// TIA Portal V19 program export: 12 tag tables, 4 data types, 5 data blocks, 16 code blocks (in call order from the OBs), 12 instance data blocks

VAR_GLOBAL   // PLC tag table "Default tag table"
   FirstScan AT %M101.0 : Bool;
   DiagStatusUpdate AT %M101.1 : Bool;
   AlwaysTRUE AT %M101.2 : Bool;
   AlwaysFALSE AT %M101.3 : Bool;
   System_Byte AT %MB101 : Byte;
   Clock_Byte AT %MB100 : Byte;
   Clock_10Hz AT %M100.0 : Bool;
   Clock_5Hz AT %M100.1 : Bool;
   "Clock_2.5Hz" AT %M100.2 : Bool;
   Clock_2Hz AT %M100.3 : Bool;
   "Clock_1.25Hz" AT %M100.4 : Bool;
   Clock_1Hz AT %M100.5 : Bool;
   "Clock_0.625Hz" AT %M100.6 : Bool;
   "Clock_0.5Hz" AT %M100.7 : Bool;
END_VAR

VAR_GLOBAL   // PLC tag table "DemoCaseTags"
   POT4_G120 AT %MD30 : Real;
   HMI_IO_Test AT %M10.4 : Bool;
   PB_Green_1200 AT %M60.0 : Bool;
   PB_Blue_1200 AT %M60.1 : Bool;
   POT3_Upper_1200 AT %MW62 : Int;
   PB_Green_Lamp_1200 AT %M64.0 : Bool;
   PB_Blue_Lamp_1200 AT %M64.1 : Bool;
   TopLights_Green_1200 AT %M64.5 : Bool;
   TopLights_Red_1200 AT %M64.6 : Bool;
   TopLights_Blue_1200 AT %M64.7 : Bool;
   "1200_Inputs" AT %MB60 : Byte;
   "1200_Outputs" AT %MB64 : Byte;
   "1200_All_Inputs" AT %MD60 : DWord;
   OS6 AT %M11.4 : Bool;
   "Red Latch" AT %M11.5 : Bool;
   "Green Latch" AT %M11.6 : Bool;
   GateClosed AT %M11.7 : Bool;
   "Blue Latch" AT %M20.3 : Bool;
   Coordination AT %MW36 : Int;
   POT2_Warning AT %M20.4 : Bool;
END_VAR

VAR_GLOBAL   // PLC tag table "HMIConveyor"
   ConveyorOn AT %M10.0 : Bool;
   ConveyorMoving AT %M10.1 : Bool;
   Conveyor_MPM AT %MW12 : Int;
   Conveyor_Max_MPM AT %MW14 : Int;
   Start_System_HMI AT %M20.0 : Bool;
   Stop_System_HMI AT %M20.1 : Bool;
   Reset_System_HMI AT %M20.2 : Bool;
   OS1 AT %M10.2 : Bool;
   ARM_MPM AT %MW34 : Int;
   OS11 AT %M74.3 : Bool;
END_VAR

VAR_GLOBAL   // PLC tag table "KP8Tags"
   Toggle_Switch2 AT %M50.0 : Bool;   // KP8 bit that is toggled each time is pressed
   HMI_KP8_JogFwd AT %M50.1 : Bool;
   HMI_KP8_Stop AT %M50.2 : Bool;
   Toggle_Switch1 AT %M50.4 : Bool;   // KP8 bit that is toggled each time is pressed
   HMI_KP8_JogRev AT %M50.5 : Bool;
   HMI_KP8_Start AT %M50.6 : Bool;
   Toggle_Enable_Disable AT %M50.7 : Bool;   // KP8 bit that is toggled each time is pressed
   HMI_KP8_Red AT %MB70 : Byte;
   HMI_KP8_Green AT %MB71 : Byte;
   HMI_KP8_Blue AT %MB72 : Byte;
   HMI_KP8_Enable_Disable AT %M73.0 : Bool;
   HMI_KP8_Reset AT %M73.1 : Bool;
   HMI_KP8_Switch1 AT %M73.2 : Bool;
   HMI_KP8_Switch2 AT %M73.3 : Bool;
   OS8 AT %M74.0 : Bool;
   OS9 AT %M74.1 : Bool;
   OS10 AT %M74.2 : Bool;
END_VAR

VAR_GLOBAL   // PLC tag table "SafetyTags"
   Safety_PB_Blue_Lamp AT %M90.0 : Bool;
END_VAR

VAR_GLOBAL   // PLC tag table "Speed Control"
   POT2_Lower_Real AT %MD38 : Real;
   Tmp AT %MW4 : Word;
   POT1_Upper__Real AT %MD16 : Real;
   MyIndex AT %MW6 : Int;
   Drive_Error AT %M11.3 : Bool;
   OS2 AT %M10.3 : Bool;
   OS3 AT %M10.5 : Bool;
   G120_Error AT %M10.6 : Bool;
   G120_Enabled AT %M10.7 : Bool;
   G120_Run_Velocity AT %M11.0 : Bool;
   OS4 AT %M11.1 : Bool;
   OS5 AT %M11.2 : Bool;
   BusyMV AT %M0.0 : Bool;
   OS7 AT %M21.3 : Bool;
   ConveyorWorking AT %M6.0 : Bool;   // Conveyor Diagnostic Tag
END_VAR

VAR_GLOBAL   // PLC tag table "Encoder"
END_VAR

VAR_GLOBAL   // PLC tag table "G120"
   SpeedAxis_1_Actor_Interface_AddressIn AT %I256.0 : "PD_TEL1_IN";
   SpeedAxis_1_Actor_Interface_AddressOut AT %Q256.0 : "PD_TEL1_OUT";
END_VAR

VAR_GLOBAL   // PLC tag table "KP8"
   Jog_Reverse_Green_KP8 AT %Q51.5 : Bool;   // KP8
   Enable_Disable_KP8 AT %I50.7 : Bool;   // KP8
   Drive_Start_KP8 AT %I50.6 : Bool;   // KP8
   Jog_Reverse_KP8 AT %I50.5 : Bool;   // KP8
   Switch1_KP8 AT %I50.4 : Bool;   // KP8
   Enable_Disable_Green_KP8 AT %Q51.7 : Bool;   // KP8
   Drive_Start_Red_KP8 AT %Q50.6 : Bool;   // KP8
   Jog_Reverse_Red_KP8 AT %Q50.5 : Bool;   // KP8
   Switch1_Red_KP8 AT %Q50.4 : Bool;   // KP8
   RESET_KP8 AT %I50.3 : Bool;   // KP8
   Drive_Stop_KP8 AT %I50.2 : Bool;   // KP8
   Jog_Forward_KP8 AT %I50.1 : Bool;   // KP8
   RESET_Red_KP8 AT %Q50.3 : Bool;   // KP8
   Drive_Stop_Red_KP8 AT %Q50.2 : Bool;   // KP8
   Jog_Forward_Red_KP8 AT %Q50.1 : Bool;   // KP8
   Switch2_KP8 AT %I50.0 : Bool;   // KP8
   Switch2_Red_KP8 AT %Q50.0 : Bool;   // KP8
   Enable_Disable_Red_KP8 AT %Q50.7 : Bool;   // KP8
   Drive_Start_Green_KP8 AT %Q51.6 : Bool;   // KP8
   Switch1_Green_KP8 AT %Q51.4 : Bool;   // KP8
   RESET_Green_KP8 AT %Q51.3 : Bool;   // KP8
   Drive_Stop_Green_KP8 AT %Q51.2 : Bool;   // KP8
   Jog_Forward_Green_KP8 AT %Q51.1 : Bool;   // KP8
   Switch2_Green_KP8 AT %Q51.0 : Bool;   // KP8
   Switch2_Blue_KP8 AT %Q52.0 : Bool;   // KP8
   Jog_Forward_Blue_KP8 AT %Q52.1 : Bool;   // KP8
   Drive_Stop_Blue_KP8 AT %Q52.2 : Bool;   // KP8
   RESET_Blue_KP8 AT %Q52.3 : Bool;   // KP8
   Switch1_Blue_KP8 AT %Q52.4 : Bool;   // KP8
   Jog_Reverse_Blue_KP8 AT %Q52.5 : Bool;   // KP8
   Drive_Start_Blue_KP8 AT %Q52.6 : Bool;   // KP8
   Enable_Disable_Blue_KP8 AT %Q52.7 : Bool;   // KP8
   KP8_Red AT %QB50 : Byte;   // KP8
   KP8_Green AT %QB51 : Byte;   // KP8
   KP8_Blue AT %QB52 : Byte;   // KP8
END_VAR

VAR_GLOBAL   // PLC tag table "LocalMP"
   PB_Green_1500 AT %I0.0 : Bool;
   PB_Blue_1500 AT %I0.1 : Bool;
   POT1_Upper_1500 AT %IW6 : Int;   // connected to AI channel 2
   POT2_Lower_1500 AT %IW14 : Int;   // connected to AI channel 6
END_VAR

VAR_GLOBAL   // PLC tag table "RemoteSP"
   PB_Green_Lamp AT %Q8.0 : Bool;
   PB_Blue_Lamp AT %Q8.1 : Bool;
   TopLights_green_1500 AT %Q10.0 : Bool;   // TopLight green 1=on 0=off
   TopLights_red_1500 AT %Q10.1 : Bool;   // TopLight red 1=on 0=off
   TopLights_blue_1500 AT %Q10.2 : Bool;   // TopLight blue 1=on 0=off
   "ESTOP CH1" AT %I18.1 : Bool;
   Estop_LED AT %Q24.0 : Bool;
   "RFID_Gate CH1" AT %I18.0 : Bool;
   RFID_Gate_AUX AT %I22.2 : Bool;
END_VAR

VAR_GLOBAL   // PLC tag table "S71200IDevice"
   "Out to 1200" AT %QW100 : Int;
   PB_Green_from_1200 AT %I100.0 : Bool;
   PB_Blue_from_1200 AT %I100.1 : Bool;
   POT_from_1200 AT %IW102 : Word;
END_VAR

TYPE "HEADER"
   STRUCT
      REQ_REF : Byte;
      REQ_ID : Byte;
      AXIS : Byte;
      NO_PARAM : Byte;
   END_STRUCT;
END_TYPE

TYPE "PARAMETERADDR"
   STRUCT
      ATTRIBUTE : Byte;
      NO_ELEM : Byte;
      PARA_NO : Word;
      SUBINDEX : Word;
   END_STRUCT;
END_TYPE

TYPE "SiemensDataType"
   STRUCT
      Test1 : Bool;
      Test2 : Bool;
      Test3 : Bool;
      Test4 : Bool;
      Test5 : Bool;
      Test6 : Bool;
      Test7 : Bool;
   END_STRUCT;
END_TYPE

TYPE "Time Zone"
   STRUCT
      City : String;
      "Local Time" : Time_Of_Day;
      Offset : Time;
   END_STRUCT;
END_TYPE

DATA_BLOCK "GlobalDB"   // DB2
{ S7_Optimized_Access := 'TRUE' }
// stored: MemoryReserve 100
   VAR
      TagData : "SiemensDataType";
   END_VAR
BEGIN
END_DATA_BLOCK

DATA_BLOCK "GraphicsData"   // DB1
{ S7_Optimized_Access := 'TRUE' }
// stored: MemoryReserve 100
   VAR
      HMI_Graphic_Index : Int;
      HMI_Box_Cnt : DInt;
      HMI_Pallet_Cnt : DInt;
   END_VAR
BEGIN
END_DATA_BLOCK

DATA_BLOCK "TimeZones"   // DB13
{ S7_Optimized_Access := 'TRUE' }
// stored: MemoryReserve 100
   VAR
      UTC_0 : "Time Zone";
      UTC_1 { S7_SetPoint := 'True'} : "Time Zone";
      UTC_2 { S7_SetPoint := 'True'} : "Time Zone";
   END_VAR
BEGIN
   UTC_0.City := 'London';
   UTC_0.Offset := T#0H;
   UTC_1.City := 'Berlin';
   UTC_1.Offset := T#1H;
   UTC_2.City := 'Cairo';
   UTC_2.Offset := T#2H;
END_DATA_BLOCK

DATA_BLOCK "TestInterConnLPythagorean"   // DB10001
{ S7_Optimized_Access := 'TRUE' }
// #@AutoGenerated
// stored: MemoryReserve 100
   VAR
      "a" : Real;
      "b" : Real;
      c : Real;
      valid : Bool;
   END_VAR
BEGIN
END_DATA_BLOCK

DATA_BLOCK "Connect_DB"   // DB7
{ S7_Optimized_Access := 'TRUE' }
// stored: MemoryReserve 100
   VAR
      "Out to 1200" : Int;
   END_VAR
BEGIN
END_DATA_BLOCK

ORGANIZATION_BLOCK "Main"   // OB1, LAD, ProgramCycle
TITLE = "Main Program Sweep (Cycle)"
{ S7_Optimized_Access := 'TRUE' }
// TIA Demo Project
// 1500 password is Siemens1
// stored: SetENOAutomatically false
   VAR_INPUT
      Initial_Call : Bool;   // Initial call of this OB
      Remanence : Bool;   // =True, if remanent data are available
   END_VAR
   VAR_TEMP   // added for the SCL form of the ladder/FBD networks
      _w1 : Bool;
      _w2 : Bool;
   END_VAR
BEGIN

REGION Network 1: Scale the Potentiometer raw value to a Real between 0.0-1500.0
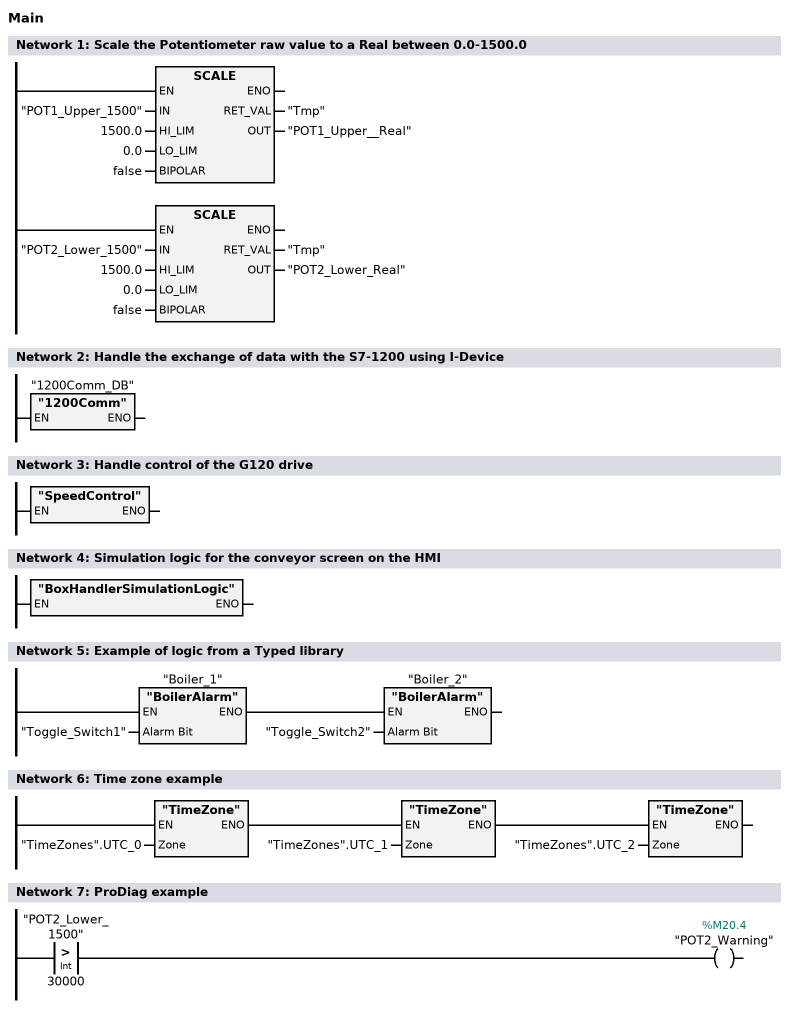
   "Tmp" := SCALE(IN := "POT1_Upper_1500",
                  HI_LIM := 1500.0,
                  LO_LIM := 0.0,
                  BIPOLAR := false,
                  OUT => "POT1_Upper__Real");
   "Tmp" := SCALE(IN := "POT2_Lower_1500",
                  HI_LIM := 1500.0,
                  LO_LIM := 0.0,
                  BIPOLAR := false,
                  OUT => "POT2_Lower_Real");
END_REGION

REGION Network 2: Handle the exchange of data with the S7-1200 using I-Device
   RUNG wire#powerrail
      "1200Comm_DB"()
   END_RUNG
   // the same network as SCL:
   "1200Comm_DB"();   // "1200Comm"
END_REGION

REGION Network 3: Handle control of the G120 drive
   RUNG wire#powerrail
      "SpeedControl"()
   END_RUNG
   // the same network as SCL:
   "SpeedControl"();
END_REGION

REGION Network 4: Simulation logic for the conveyor screen on the HMI
   RUNG wire#powerrail
      "BoxHandlerSimulationLogic"()
   END_RUNG
   // the same network as SCL:
   "BoxHandlerSimulationLogic"();
END_REGION

REGION Network 5: Example of logic from a Typed library
   RUNG wire#powerrail
      "Boiler_1"("Alarm Bit" := "Toggle_Switch1")
      "Boiler_2"("Alarm Bit" := "Toggle_Switch2")
   END_RUNG
   // the same network as SCL:
   "Boiler_1"("Alarm Bit" := "Toggle_Switch1", ENO => #_w1);   // "BoilerAlarm"
   IF #_w1 THEN
       "Boiler_2"("Alarm Bit" := "Toggle_Switch2");   // "BoilerAlarm"
   END_IF;
END_REGION

REGION Network 6: Time zone example
   RUNG wire#powerrail
      "TimeZone"(Zone := "TimeZones".UTC_0)
      "TimeZone"(Zone := "TimeZones".UTC_1)
      "TimeZone"(Zone := "TimeZones".UTC_2)
   END_RUNG
   // the same network as SCL:
   "TimeZone"(Zone := "TimeZones".UTC_0, ENO => #_w1);
   "TimeZone"(EN := #_w1, Zone := "TimeZones".UTC_1, ENO => #_w2);
   IF #_w2 THEN "TimeZone"(Zone := "TimeZones".UTC_2); END_IF;
END_REGION

REGION Network 7: ProDiag example
   RUNG wire#powerrail
      { S7_Templates := "SrcType := Int" } GT_Contact(in1 := "POT2_Lower_1500", in2 := 30000)
      Coil( "POT2_Warning" )
   END_RUNG
   // the same network as SCL:
   "POT2_Warning" := "POT2_Lower_1500" > 30000;
END_REGION
END_ORGANIZATION_BLOCK

FUNCTION_BLOCK "1200Comm"   // FB3, LAD
TITLE = I Device exchange of data with the S7-1200
{ S7_Optimized_Access := 'TRUE' }
// stored: MemoryReserve 100, SetENOAutomatically false
BEGIN

REGION Network 1: Pass light data to the 1200
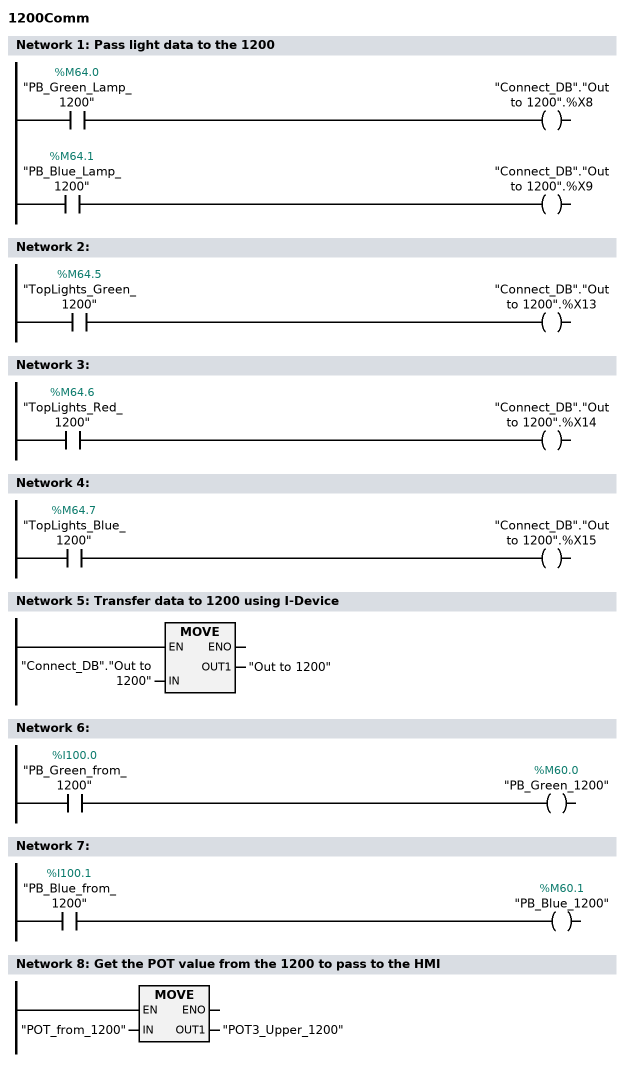
   RUNG wire#powerrail
      Contact( "PB_Green_Lamp_1200" )
      Coil( "Connect_DB"."Out to 1200".%X8 )
   END_RUNG
   RUNG wire#powerrail
      Contact( "PB_Blue_Lamp_1200" )
      Coil( "Connect_DB"."Out to 1200".%X9 )
   END_RUNG
   // the same network as SCL:
   "Connect_DB"."Out to 1200".%X8 := "PB_Green_Lamp_1200";
   "Connect_DB"."Out to 1200".%X9 := "PB_Blue_Lamp_1200";
END_REGION

REGION Network 2
   RUNG wire#powerrail
      Contact( "TopLights_Green_1200" )
      Coil( "Connect_DB"."Out to 1200".%X13 )
   END_RUNG
   // the same network as SCL:
   "Connect_DB"."Out to 1200".%X13 := "TopLights_Green_1200";
END_REGION

REGION Network 3
   RUNG wire#powerrail
      Contact( "TopLights_Red_1200" )
      Coil( "Connect_DB"."Out to 1200".%X14 )
   END_RUNG
   // the same network as SCL:
   "Connect_DB"."Out to 1200".%X14 := "TopLights_Red_1200";
END_REGION

REGION Network 4
   RUNG wire#powerrail
      Contact( "TopLights_Blue_1200" )
      Coil( "Connect_DB"."Out to 1200".%X15 )
   END_RUNG
   // the same network as SCL:
   "Connect_DB"."Out to 1200".%X15 := "TopLights_Blue_1200";
END_REGION

REGION Network 5: Transfer data to 1200 using I-Device
   RUNG wire#powerrail
      Move(in := "Connect_DB"."Out to 1200", out1 => "Out to 1200")
   END_RUNG
   // the same network as SCL:
   "Out to 1200" := "Connect_DB"."Out to 1200";
END_REGION

REGION Network 6
   RUNG wire#powerrail
      Contact( "PB_Green_from_1200" )
      Coil( "PB_Green_1200" )
   END_RUNG
   // the same network as SCL:
   "PB_Green_1200" := "PB_Green_from_1200";
END_REGION

REGION Network 7
   RUNG wire#powerrail
      Contact( "PB_Blue_from_1200" )
      Coil( "PB_Blue_1200" )
   END_RUNG
   // the same network as SCL:
   "PB_Blue_1200" := "PB_Blue_from_1200";
END_REGION

REGION Network 8: Get the POT value from the 1200 to pass to the HMI
   RUNG wire#powerrail
      Move(in := "POT_from_1200", out1 => "POT3_Upper_1200")
   END_RUNG
   // the same network as SCL:
   "POT3_Upper_1200" := "POT_from_1200";
END_REGION
END_FUNCTION_BLOCK

FUNCTION "SpeedControl" : Void   // FC1, LAD
TITLE = G120 drive Control
{ S7_Optimized_Access := 'TRUE' }
// stored: SetENOAutomatically false
   VAR_TEMP   // added for the SCL form of the ladder/FBD networks
      _w1 : Bool;
      _w2 : Bool;
   END_VAR
BEGIN

REGION Network 1: Enable the G120
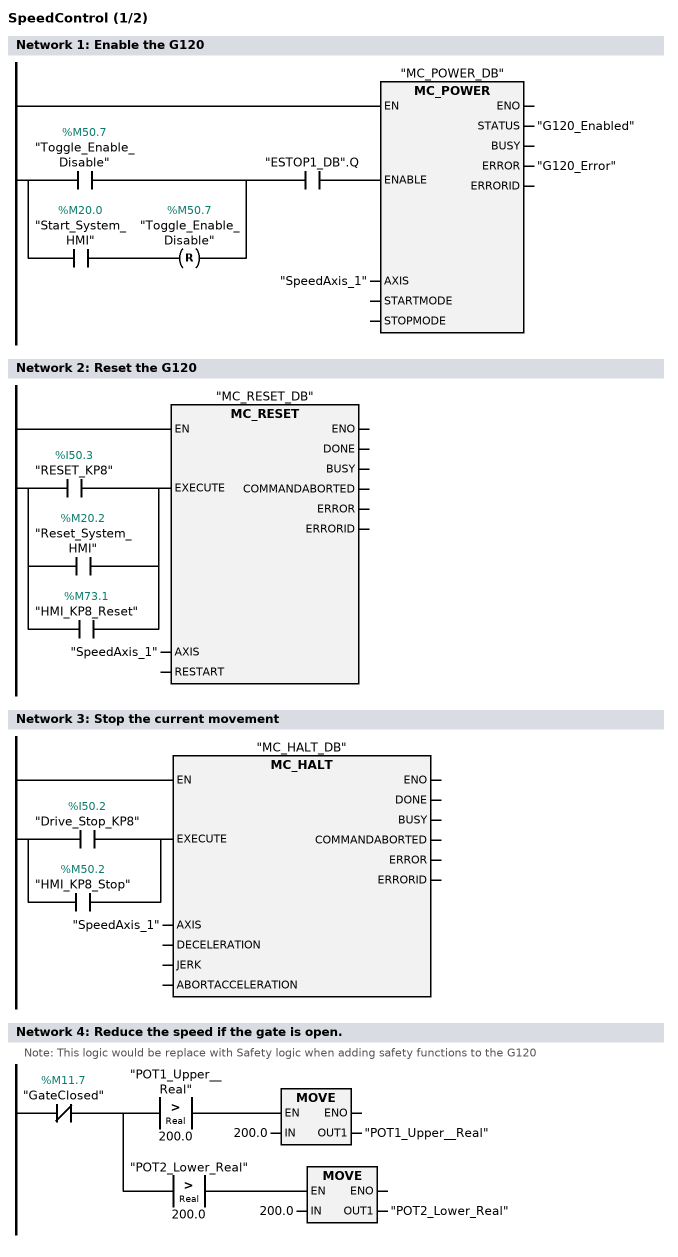
   RUNG wire#powerrail
      "MC_POWER_DB".MC_POWER(Enable := wire#w2, Axis := "SpeedAxis_1", StartMode :=, StopMode :=, Status => "G120_Enabled", Busy =>, Error => "G120_Error", ErrorId =>)
   END_RUNG
   RUNG wire#powerrail
      Contact( "Toggle_Enable_Disable" )
      wire#w1
      Contact( "ESTOP1_DB".Q )
   END_RUNG wire#w2
   RUNG wire#powerrail
      Contact( "Start_System_HMI" )
      R_Coil( "Toggle_Enable_Disable" )
   END_RUNG wire#w1
   // the same network as SCL:
   #_w1 := "Toggle_Enable_Disable";
   IF "Start_System_HMI" THEN "Toggle_Enable_Disable" := FALSE; END_IF;
   "MC_POWER_DB"(Enable := (#_w1 OR "Start_System_HMI") AND "ESTOP1_DB".Q,   // MC_POWER
                 Axis := "SpeedAxis_1",
                 Status => "G120_Enabled",
                 Error => "G120_Error");
END_REGION

REGION Network 2: Reset the G120
   RUNG wire#powerrail
      "MC_RESET_DB".MC_RESET(Execute := wire#w1, Axis := "SpeedAxis_1", Restart :=, Done =>, Busy =>, CommandAborted =>, Error =>, ErrorId =>)
   END_RUNG
   RUNG wire#powerrail
      Contact( "RESET_KP8" )
   END_RUNG wire#w1
   RUNG wire#powerrail
      Contact( "Reset_System_HMI" )
   END_RUNG wire#w1
   RUNG wire#powerrail
      Contact( "HMI_KP8_Reset" )
   END_RUNG wire#w1
   // the same network as SCL:
   "MC_RESET_DB"(Execute := "RESET_KP8" OR "Reset_System_HMI" OR "HMI_KP8_Reset", Axis := "SpeedAxis_1");   // MC_RESET
END_REGION

REGION Network 3: Stop the current movement
   RUNG wire#powerrail
      "MC_HALT_DB".MC_HALT(Execute := wire#w1, Axis := "SpeedAxis_1", Deceleration :=, Jerk :=, AbortAcceleration :=, Done =>, Busy =>, CommandAborted =>, Error =>, ErrorId =>)
   END_RUNG
   RUNG wire#powerrail
      Contact( "Drive_Stop_KP8" )
   END_RUNG wire#w1
   RUNG wire#powerrail
      Contact( "HMI_KP8_Stop" )
   END_RUNG wire#w1
   // the same network as SCL:
   "MC_HALT_DB"(Execute := "Drive_Stop_KP8" OR "HMI_KP8_Stop", Axis := "SpeedAxis_1");   // MC_HALT
END_REGION

REGION Network 4: Reduce the speed if the gate is open.
   // Note: This logic would be replace with Safety logic when adding safety functions to the G120
   RUNG wire#powerrail
      I_Contact( "GateClosed" )
      wire#w1
      { S7_Templates := "SrcType := Real" } GT_Contact(in1 := "POT1_Upper__Real", in2 := 200.0)
      Move(in := 200.0, out1 => "POT1_Upper__Real")
   END_RUNG
   RUNG wire#w1
      { S7_Templates := "SrcType := Real" } GT_Contact(in1 := "POT2_Lower_Real", in2 := 200.0)
      Move(in := 200.0, out1 => "POT2_Lower_Real")
   END_RUNG
   // the same network as SCL:
   IF NOT "GateClosed" AND ("POT1_Upper__Real" > 200.0) THEN "POT1_Upper__Real" := 200.0; END_IF;
   IF NOT "GateClosed" AND ("POT2_Lower_Real" > 200.0) THEN "POT2_Lower_Real" := 200.0; END_IF;
END_REGION

REGION Network 5: Move at a constant velocity
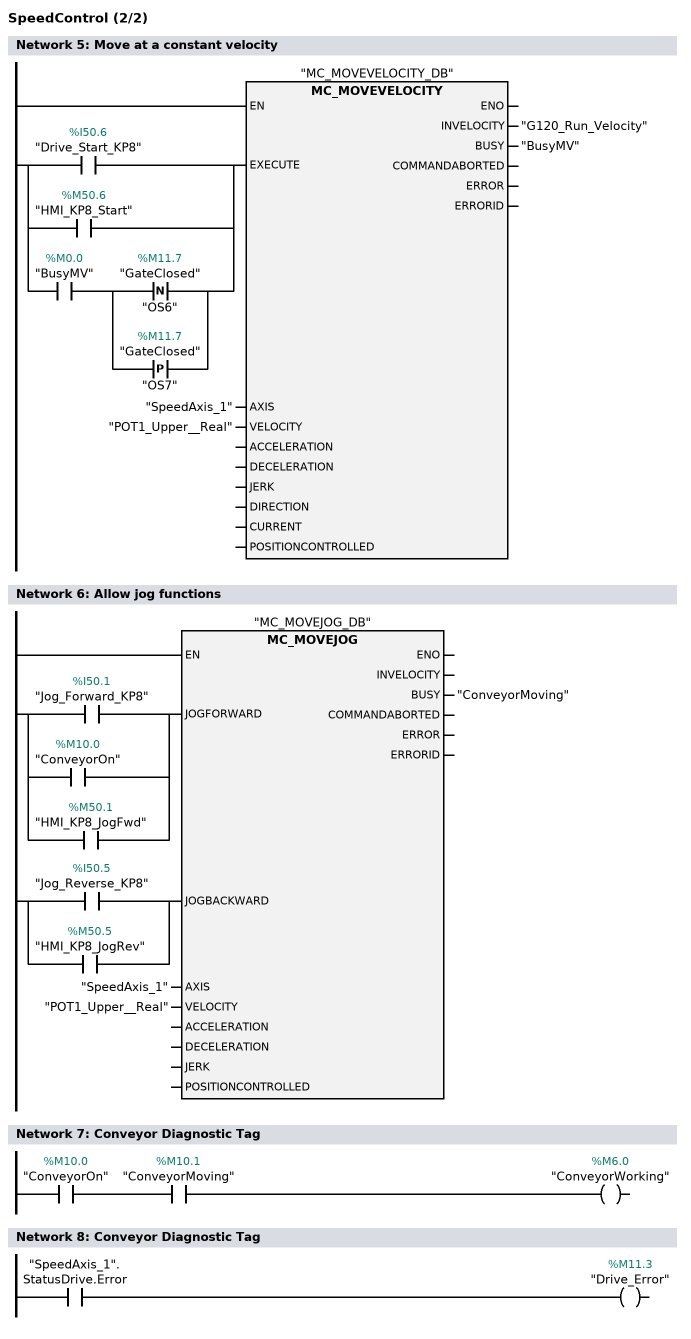
   RUNG wire#powerrail
      "MC_MOVEVELOCITY_DB".MC_MOVEVELOCITY(Execute := wire#w2, Axis := "SpeedAxis_1", Velocity := "POT1_Upper__Real", Acceleration :=, Deceleration :=, Jerk :=, Direction :=, Current :=, PositionControlled :=, InVelocity => "G120_Run_Velocity", Busy => "BusyMV", CommandAborted =>, Error =>, ErrorId =>)
   END_RUNG
   RUNG wire#powerrail
      Contact( "Drive_Start_KP8" )
   END_RUNG wire#w2
   RUNG wire#powerrail
      Contact( "HMI_KP8_Start" )
   END_RUNG wire#w2
   RUNG wire#powerrail
      Contact( "BusyMV" )
      wire#w1
      N_Contact(operand := "GateClosed", bit := "OS6")
   END_RUNG wire#w2
   RUNG wire#w1
      P_Contact(operand := "GateClosed", bit := "OS7")
   END_RUNG wire#w2
   // the same network as SCL:
   #_w1 := "BusyMV" AND NOT "GateClosed" AND "OS6";   // falling edge of "GateClosed"
   "OS6" := "GateClosed";
   #_w2 := "BusyMV" AND "GateClosed" AND NOT "OS7";   // rising edge of "GateClosed"
   "OS7" := "GateClosed";
   "MC_MOVEVELOCITY_DB"(Execute := "Drive_Start_KP8" OR "HMI_KP8_Start" OR #_w1 OR #_w2,   // MC_MOVEVELOCITY
                        Axis := "SpeedAxis_1",
                        Velocity := "POT1_Upper__Real",
                        InVelocity => "G120_Run_Velocity",
                        Busy => "BusyMV");
END_REGION

REGION Network 6: Allow jog functions
   RUNG wire#powerrail
      "MC_MOVEJOG_DB".MC_MOVEJOG(JogForward := wire#w1, JogBackward := wire#w2, Axis := "SpeedAxis_1", Velocity := "POT1_Upper__Real", Acceleration :=, Deceleration :=, Jerk :=, PositionControlled :=, InVelocity =>, Busy => "ConveyorMoving", CommandAborted =>, Error =>, ErrorId =>)
   END_RUNG
   RUNG wire#powerrail
      Contact( "Jog_Forward_KP8" )
   END_RUNG wire#w1
   RUNG wire#powerrail
      Contact( "ConveyorOn" )
   END_RUNG wire#w1
   RUNG wire#powerrail
      Contact( "HMI_KP8_JogFwd" )
   END_RUNG wire#w1
   RUNG wire#powerrail
      Contact( "Jog_Reverse_KP8" )
   END_RUNG wire#w2
   RUNG wire#powerrail
      Contact( "HMI_KP8_JogRev" )
   END_RUNG wire#w2
   // the same network as SCL:
   "MC_MOVEJOG_DB"(JogForward := "Jog_Forward_KP8" OR "ConveyorOn" OR "HMI_KP8_JogFwd",   // MC_MOVEJOG
                   JogBackward := "Jog_Reverse_KP8" OR "HMI_KP8_JogRev",
                   Axis := "SpeedAxis_1",
                   Velocity := "POT1_Upper__Real",
                   Busy => "ConveyorMoving");
END_REGION

REGION Network 7: Conveyor Diagnostic Tag
   RUNG wire#powerrail
      Contact( "ConveyorOn" )
      Contact( "ConveyorMoving" )
      Coil( "ConveyorWorking" )
   END_RUNG
   // the same network as SCL:
   "ConveyorWorking" := "ConveyorOn" AND "ConveyorMoving";
END_REGION

REGION Network 8: Conveyor Diagnostic Tag
   RUNG wire#powerrail
      Contact( "SpeedAxis_1".StatusDrive.Error )
      Coil( "Drive_Error" )
   END_RUNG
   // the same network as SCL:
   "Drive_Error" := "SpeedAxis_1".StatusDrive.Error;
END_REGION
END_FUNCTION

FUNCTION "BoxHandlerSimulationLogic" : Void   // FC20, LAD
{ S7_Optimized_Access := 'TRUE' }
// stored: AutoNumber false, SetENOAutomatically false
   VAR_TEMP
      ArmOn : Bool;
      ArmSpeed : Real;
   END_VAR
   VAR_TEMP   // added for the SCL form of the ladder/FBD networks
      _w1 : Bool;
      _w2 : Bool;
      _w3 : Bool;
   END_VAR
BEGIN

REGION Network 1: HMI Conveyor control logic
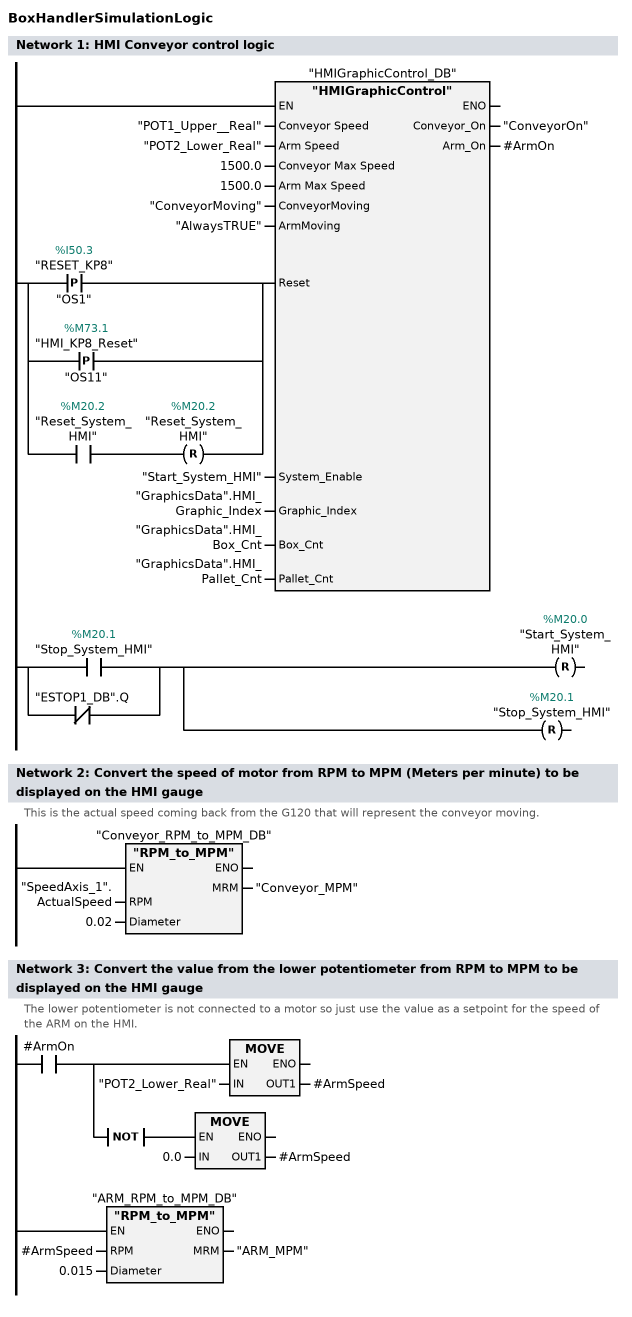
   RUNG wire#powerrail
      "HMIGraphicControl_DB"(Reset := wire#w1, "Conveyor Speed" := "POT1_Upper__Real", "Arm Speed" := "POT2_Lower_Real", "Conveyor Max Speed" := 1500.0, "Arm Max Speed" := 1500.0, ConveyorMoving := "ConveyorMoving", ArmMoving := "AlwaysTRUE", System_Enable := "Start_System_HMI", Graphic_Index := "GraphicsData".HMI_Graphic_Index, Box_Cnt := "GraphicsData".HMI_Box_Cnt, Pallet_Cnt := "GraphicsData".HMI_Pallet_Cnt, Conveyor_On => "ConveyorOn", Arm_On => #ArmOn)
   END_RUNG
   RUNG wire#powerrail
      P_Contact(operand := "RESET_KP8", bit := "OS1")
   END_RUNG wire#w1
   RUNG wire#powerrail
      P_Contact(operand := "HMI_KP8_Reset", bit := "OS11")
   END_RUNG wire#w1
   RUNG wire#powerrail
      Contact( "Reset_System_HMI" )
      R_Coil( "Reset_System_HMI" )
   END_RUNG wire#w1
   RUNG wire#powerrail
      Contact( "Stop_System_HMI" )
      wire#w2
      R_Coil( "Start_System_HMI" )
   END_RUNG
   RUNG wire#powerrail
      I_Contact( "ESTOP1_DB".Q )
   END_RUNG wire#w2
   RUNG wire#w2
      R_Coil( "Stop_System_HMI" )
   END_RUNG
   // the same network as SCL:
   #_w1 := "RESET_KP8" AND NOT "OS1";   // rising edge of "RESET_KP8"
   "OS1" := "RESET_KP8";
   #_w2 := "HMI_KP8_Reset" AND NOT "OS11";   // rising edge of "HMI_KP8_Reset"
   "OS11" := "HMI_KP8_Reset";
   #_w3 := "Reset_System_HMI";
   IF #_w3 THEN "Reset_System_HMI" := FALSE; END_IF;
   "HMIGraphicControl_DB"("Conveyor Speed" := "POT1_Upper__Real",   // "HMIGraphicControl"
                          "Arm Speed" := "POT2_Lower_Real",
                          "Conveyor Max Speed" := 1500.0,
                          "Arm Max Speed" := 1500.0,
                          ConveyorMoving := "ConveyorMoving",
                          ArmMoving := "AlwaysTRUE",
                          Reset := #_w1 OR #_w2 OR #_w3,
                          System_Enable := "Start_System_HMI",
                          Graphic_Index := "GraphicsData".HMI_Graphic_Index,
                          Box_Cnt := "GraphicsData".HMI_Box_Cnt,
                          Pallet_Cnt := "GraphicsData".HMI_Pallet_Cnt,
                          Conveyor_On => "ConveyorOn",
                          Arm_On => #ArmOn);
   IF "Stop_System_HMI" OR NOT "ESTOP1_DB".Q THEN
       "Start_System_HMI" := FALSE;
       "Stop_System_HMI" := FALSE;
   END_IF;
END_REGION

REGION Network 2: Convert the speed of motor from RPM to MPM (Meters per minute) to be displayed on the HMI gauge
   // This is the actual speed coming back from the G120 that will represent the conveyor moving.
   RUNG wire#powerrail
      "Conveyor_RPM_to_MPM_DB"(RPM := "SpeedAxis_1".ActualSpeed, Diameter := 0.02, MRM => "Conveyor_MPM")
   END_RUNG
   // the same network as SCL:
   "Conveyor_RPM_to_MPM_DB"(RPM := "SpeedAxis_1".ActualSpeed, Diameter := 0.02, MRM => "Conveyor_MPM");   // "RPM_to_MPM"
END_REGION

REGION Network 3: Convert the value from the lower potentiometer from RPM to MPM to be displayed on the HMI gauge
   // The lower potentiometer is not connected to a motor so just use the value as a setpoint for the speed of the ARM on the HMI.
   RUNG wire#powerrail
      Contact( #ArmOn )
      wire#w1
      Move(in := "POT2_Lower_Real", out1 => #ArmSpeed)
   END_RUNG
   RUNG wire#w1
      Not()
      Move(in := 0.0, out1 => #ArmSpeed)
   END_RUNG
   RUNG wire#powerrail
      "ARM_RPM_to_MPM_DB"(RPM := #ArmSpeed, Diameter := 0.015, MRM => "ARM_MPM")
   END_RUNG
   // the same network as SCL:
   IF #ArmOn THEN #ArmSpeed := "POT2_Lower_Real"; END_IF;
   IF NOT #ArmOn THEN #ArmSpeed := 0.0; END_IF;
   "ARM_RPM_to_MPM_DB"(RPM := #ArmSpeed, Diameter := 0.015, MRM => "ARM_MPM");   // "RPM_to_MPM"
END_REGION
END_FUNCTION

FUNCTION_BLOCK "HMIGraphicControl"   // FB4, LAD
{ S7_Optimized_Access := 'TRUE' }
// stored: MemoryReserve 100, SetENOAutomatically false
   VAR_INPUT
      "Conveyor Speed" { ExternalAccessible := 'False'; ExternalVisible := 'False'; ExternalWritable := 'False'} : Real;   // m/min
      "Arm Speed" { ExternalAccessible := 'False'; ExternalVisible := 'False'; ExternalWritable := 'False'} : Real;   // m/min
      "Conveyor Max Speed" { ExternalAccessible := 'False'; ExternalVisible := 'False'; ExternalWritable := 'False'} : Real := 3000.0;
      "Arm Max Speed" { ExternalAccessible := 'False'; ExternalVisible := 'False'; ExternalWritable := 'False'} : Real := 32000.0;
      ConveyorMoving : Bool := true;
      ArmMoving : Bool := true;
      Reset : Bool;
   END_VAR
   VAR_OUTPUT
      Conveyor_On : Bool;
      Arm_On : Bool;
   END_VAR
   VAR_IN_OUT
      System_Enable : Bool;
      Graphic_Index { ExternalAccessible := 'False'; ExternalVisible := 'False'; ExternalWritable := 'False'} : Int;
      Box_Cnt : DInt;
      Pallet_Cnt : DInt;
   END_VAR
   VAR
      IEC_Timer_0_Instance { S7_SetPoint := 'True'} : IEC_TIMER;
      ConveyorTick : Bool;
      ConveyorTime : DInt;
      ConveyorTimeFactor : DInt := 100000;
      ArmTick : Bool;
      ArmTimeFactor : DInt := 100000;
      ArmTime : DInt;
      IEC_Timer_0_Instance_1 { S7_SetPoint := 'True'} : IEC_TIMER;
   END_VAR
   VAR_TEMP
      ConveyorScaled : Real;
      ConveyMotor : Bool;
      ArmScaled : Real;
   END_VAR
   VAR_TEMP   // added for the SCL form of the ladder/FBD networks
      _w1 : Bool;
   END_VAR
BEGIN

REGION Network 1
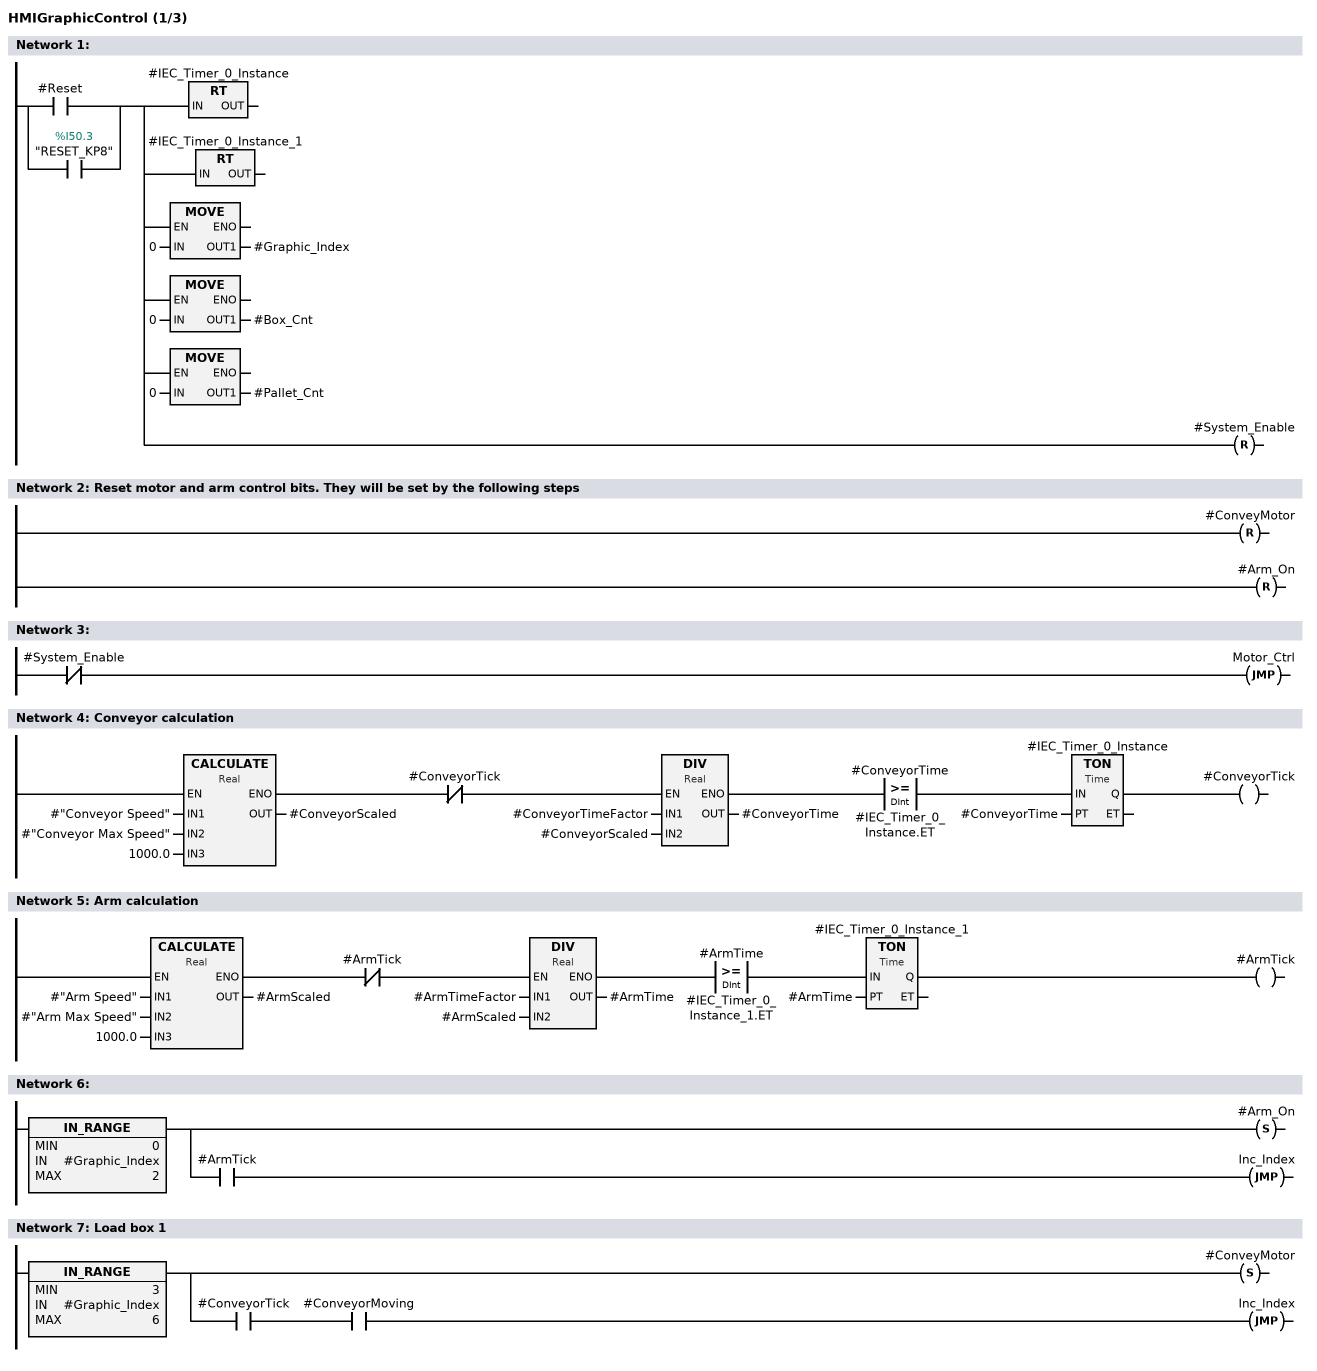
   RUNG wire#powerrail
      Contact( #Reset )
      wire#w1
      RT_Coil( #IEC_Timer_0_Instance )
   END_RUNG
   RUNG wire#powerrail
      Contact( "RESET_KP8" )
   END_RUNG wire#w1
   RUNG wire#w1
      RT_Coil( #IEC_Timer_0_Instance_1 )
   END_RUNG
   RUNG wire#w1
      Move(in := 0, out1 => #Graphic_Index)
   END_RUNG
   RUNG wire#w1
      Move(in := 0, out1 => #Box_Cnt)
   END_RUNG
   RUNG wire#w1
      Move(in := 0, out1 => #Pallet_Cnt)
   END_RUNG
   RUNG wire#w1
      R_Coil( #System_Enable )
   END_RUNG
   // the same network as SCL:
   #_w1 := #Reset OR "RESET_KP8";
   IF #_w1 THEN
       RESET_TIMER(#IEC_Timer_0_Instance);
       RESET_TIMER(#IEC_Timer_0_Instance_1);
       #Graphic_Index := 0;
       #Box_Cnt := 0;
       #Pallet_Cnt := 0;
       #System_Enable := FALSE;
   END_IF;
END_REGION

REGION Network 2: Reset motor and arm control bits. They will be set by the following steps
   RUNG wire#powerrail
      R_Coil( #ConveyMotor )
   END_RUNG
   RUNG wire#powerrail
      R_Coil( #Arm_On )
   END_RUNG
   // the same network as SCL:
   #ConveyMotor := FALSE;
   #Arm_On := FALSE;
END_REGION

REGION Network 3
   RUNG wire#powerrail
      I_Contact( #System_Enable )
      JumpCoil( Motor_Ctrl )
   END_RUNG
   // the same network as SCL:
   IF NOT #System_Enable THEN GOTO Motor_Ctrl; END_IF;
END_REGION

REGION Network 4: Conveyor calculation
   RUNG wire#powerrail
      { S7_Templates := "SrcType := Real"; S7_Expression := "IN1/IN2*IN3" } Calculate(in1 := #"Conveyor Speed", in2 := #"Conveyor Max Speed", in3 := 1000.0, out => #ConveyorScaled)
      I_Contact( #ConveyorTick )
      { S7_Templates := "SrcType := Real"; S7_GenerateENO := "TRUE" } Div(in1 := #ConveyorTimeFactor, in2 := #ConveyorScaled, out => #ConveyorTime)
      { S7_Templates := "SrcType := DInt" } GE_Contact(in1 := #ConveyorTime, in2 := #IEC_Timer_0_Instance.ET)
      { S7_Templates := "time_type := Time" } #IEC_Timer_0_Instance.TON(pt := #ConveyorTime, et =>)
      Coil( #ConveyorTick )
   END_RUNG
   // the same network as SCL:
   // ENO of a box is taken as its EN; it also drops when the box reports an error
   #ConveyorScaled := #"Conveyor Speed"/#"Conveyor Max Speed"*1000.0;
   IF NOT #ConveyorTick THEN #ConveyorTime := #ConveyorTimeFactor / #ConveyorScaled; END_IF;
   #IEC_Timer_0_Instance.TON(IN := NOT #ConveyorTick AND (#ConveyorTime >= #IEC_Timer_0_Instance.ET),
                           PT := #ConveyorTime);
   #ConveyorTick := #IEC_Timer_0_Instance.Q;
END_REGION

REGION Network 5: Arm calculation
   RUNG wire#powerrail
      { S7_Templates := "SrcType := Real"; S7_Expression := "IN1/IN2*IN3" } Calculate(in1 := #"Arm Speed", in2 := #"Arm Max Speed", in3 := 1000.0, out => #ArmScaled)
      I_Contact( #ArmTick )
      { S7_Templates := "SrcType := Real"; S7_GenerateENO := "TRUE" } Div(in1 := #ArmTimeFactor, in2 := #ArmScaled, out => #ArmTime)
      { S7_Templates := "SrcType := DInt" } GE_Contact(in1 := #ArmTime, in2 := #IEC_Timer_0_Instance_1.ET)
      { S7_Templates := "time_type := Time" } #IEC_Timer_0_Instance_1.TON(pt := #ArmTime, et =>)
      Coil( #ArmTick )
   END_RUNG
   // the same network as SCL:
   // ENO of a box is taken as its EN; it also drops when the box reports an error
   #ArmScaled := #"Arm Speed"/#"Arm Max Speed"*1000.0;
   IF NOT #ArmTick THEN #ArmTime := #ArmTimeFactor / #ArmScaled; END_IF;
   #IEC_Timer_0_Instance_1.TON(IN := NOT #ArmTick AND (#ArmTime >= #IEC_Timer_0_Instance_1.ET), PT := #ArmTime);
   #ArmTick := #IEC_Timer_0_Instance_1.Q;
END_REGION

REGION Network 6
   RUNG wire#powerrail
      { S7_Templates := "SrcType := Int" } InRange(min := 0, in := #Graphic_Index, max := 2)
      wire#w1
      S_Coil( #Arm_On )
   END_RUNG
   RUNG wire#w1
      Contact( #ArmTick )
      JumpCoil( Inc_Index )
   END_RUNG
   // the same network as SCL:
   #_w1 := (0 <= #Graphic_Index) AND (#Graphic_Index <= 2);
   IF #_w1 THEN #Arm_On := TRUE; END_IF;
   IF #_w1 AND #ArmTick THEN GOTO Inc_Index; END_IF;
END_REGION

REGION Network 7: Load box 1
   RUNG wire#powerrail
      { S7_Templates := "SrcType := Int" } InRange(min := 3, in := #Graphic_Index, max := 6)
      wire#w1
      S_Coil( #ConveyMotor )
   END_RUNG
   RUNG wire#w1
      Contact( #ConveyorTick )
      Contact( #ConveyorMoving )
      JumpCoil( Inc_Index )
   END_RUNG
   // the same network as SCL:
   #_w1 := (3 <= #Graphic_Index) AND (#Graphic_Index <= 6);
   IF #_w1 THEN #ConveyMotor := TRUE; END_IF;
   IF #_w1 AND #ConveyorTick AND #ConveyorMoving THEN GOTO Inc_Index; END_IF;
END_REGION

REGION Network 8
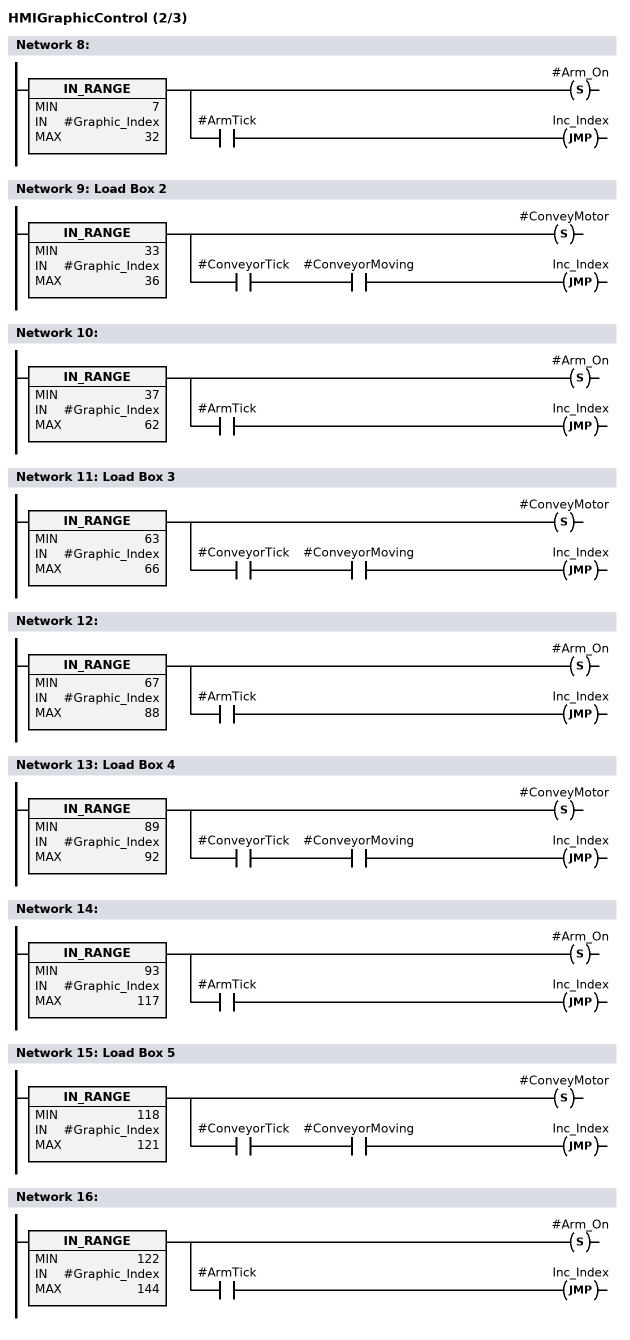
   RUNG wire#powerrail
      { S7_Templates := "SrcType := Int" } InRange(min := 7, in := #Graphic_Index, max := 32)
      wire#w1
      S_Coil( #Arm_On )
   END_RUNG
   RUNG wire#w1
      Contact( #ArmTick )
      JumpCoil( Inc_Index )
   END_RUNG
   // the same network as SCL:
   #_w1 := (7 <= #Graphic_Index) AND (#Graphic_Index <= 32);
   IF #_w1 THEN #Arm_On := TRUE; END_IF;
   IF #_w1 AND #ArmTick THEN GOTO Inc_Index; END_IF;
END_REGION

REGION Network 9: Load Box 2
   RUNG wire#powerrail
      { S7_Templates := "SrcType := Int" } InRange(min := 33, in := #Graphic_Index, max := 36)
      wire#w1
      S_Coil( #ConveyMotor )
   END_RUNG
   RUNG wire#w1
      Contact( #ConveyorTick )
      Contact( #ConveyorMoving )
      JumpCoil( Inc_Index )
   END_RUNG
   // the same network as SCL:
   #_w1 := (33 <= #Graphic_Index) AND (#Graphic_Index <= 36);
   IF #_w1 THEN #ConveyMotor := TRUE; END_IF;
   IF #_w1 AND #ConveyorTick AND #ConveyorMoving THEN GOTO Inc_Index; END_IF;
END_REGION

REGION Network 10
   RUNG wire#powerrail
      { S7_Templates := "SrcType := Int" } InRange(min := 37, in := #Graphic_Index, max := 62)
      wire#w1
      S_Coil( #Arm_On )
   END_RUNG
   RUNG wire#w1
      Contact( #ArmTick )
      JumpCoil( Inc_Index )
   END_RUNG
   // the same network as SCL:
   #_w1 := (37 <= #Graphic_Index) AND (#Graphic_Index <= 62);
   IF #_w1 THEN #Arm_On := TRUE; END_IF;
   IF #_w1 AND #ArmTick THEN GOTO Inc_Index; END_IF;
END_REGION

REGION Network 11: Load Box 3
   RUNG wire#powerrail
      { S7_Templates := "SrcType := Int" } InRange(min := 63, in := #Graphic_Index, max := 66)
      wire#w1
      S_Coil( #ConveyMotor )
   END_RUNG
   RUNG wire#w1
      Contact( #ConveyorTick )
      Contact( #ConveyorMoving )
      JumpCoil( Inc_Index )
   END_RUNG
   // the same network as SCL:
   #_w1 := (63 <= #Graphic_Index) AND (#Graphic_Index <= 66);
   IF #_w1 THEN #ConveyMotor := TRUE; END_IF;
   IF #_w1 AND #ConveyorTick AND #ConveyorMoving THEN GOTO Inc_Index; END_IF;
END_REGION

REGION Network 12
   RUNG wire#powerrail
      { S7_Templates := "SrcType := Int" } InRange(min := 67, in := #Graphic_Index, max := 88)
      wire#w1
      S_Coil( #Arm_On )
   END_RUNG
   RUNG wire#w1
      Contact( #ArmTick )
      JumpCoil( Inc_Index )
   END_RUNG
   // the same network as SCL:
   #_w1 := (67 <= #Graphic_Index) AND (#Graphic_Index <= 88);
   IF #_w1 THEN #Arm_On := TRUE; END_IF;
   IF #_w1 AND #ArmTick THEN GOTO Inc_Index; END_IF;
END_REGION

REGION Network 13: Load Box 4
   RUNG wire#powerrail
      { S7_Templates := "SrcType := Int" } InRange(min := 89, in := #Graphic_Index, max := 92)
      wire#w1
      S_Coil( #ConveyMotor )
   END_RUNG
   RUNG wire#w1
      Contact( #ConveyorTick )
      Contact( #ConveyorMoving )
      JumpCoil( Inc_Index )
   END_RUNG
   // the same network as SCL:
   #_w1 := (89 <= #Graphic_Index) AND (#Graphic_Index <= 92);
   IF #_w1 THEN #ConveyMotor := TRUE; END_IF;
   IF #_w1 AND #ConveyorTick AND #ConveyorMoving THEN GOTO Inc_Index; END_IF;
END_REGION

REGION Network 14
   RUNG wire#powerrail
      { S7_Templates := "SrcType := Int" } InRange(min := 93, in := #Graphic_Index, max := 117)
      wire#w1
      S_Coil( #Arm_On )
   END_RUNG
   RUNG wire#w1
      Contact( #ArmTick )
      JumpCoil( Inc_Index )
   END_RUNG
   // the same network as SCL:
   #_w1 := (93 <= #Graphic_Index) AND (#Graphic_Index <= 117);
   IF #_w1 THEN #Arm_On := TRUE; END_IF;
   IF #_w1 AND #ArmTick THEN GOTO Inc_Index; END_IF;
END_REGION

REGION Network 15: Load Box 5
   RUNG wire#powerrail
      { S7_Templates := "SrcType := Int" } InRange(min := 118, in := #Graphic_Index, max := 121)
      wire#w1
      S_Coil( #ConveyMotor )
   END_RUNG
   RUNG wire#w1
      Contact( #ConveyorTick )
      Contact( #ConveyorMoving )
      JumpCoil( Inc_Index )
   END_RUNG
   // the same network as SCL:
   #_w1 := (118 <= #Graphic_Index) AND (#Graphic_Index <= 121);
   IF #_w1 THEN #ConveyMotor := TRUE; END_IF;
   IF #_w1 AND #ConveyorTick AND #ConveyorMoving THEN GOTO Inc_Index; END_IF;
END_REGION

REGION Network 16
   RUNG wire#powerrail
      { S7_Templates := "SrcType := Int" } InRange(min := 122, in := #Graphic_Index, max := 144)
      wire#w1
      S_Coil( #Arm_On )
   END_RUNG
   RUNG wire#w1
      Contact( #ArmTick )
      JumpCoil( Inc_Index )
   END_RUNG
   // the same network as SCL:
   #_w1 := (122 <= #Graphic_Index) AND (#Graphic_Index <= 144);
   IF #_w1 THEN #Arm_On := TRUE; END_IF;
   IF #_w1 AND #ArmTick THEN GOTO Inc_Index; END_IF;
END_REGION

REGION Network 17: Load Box 6
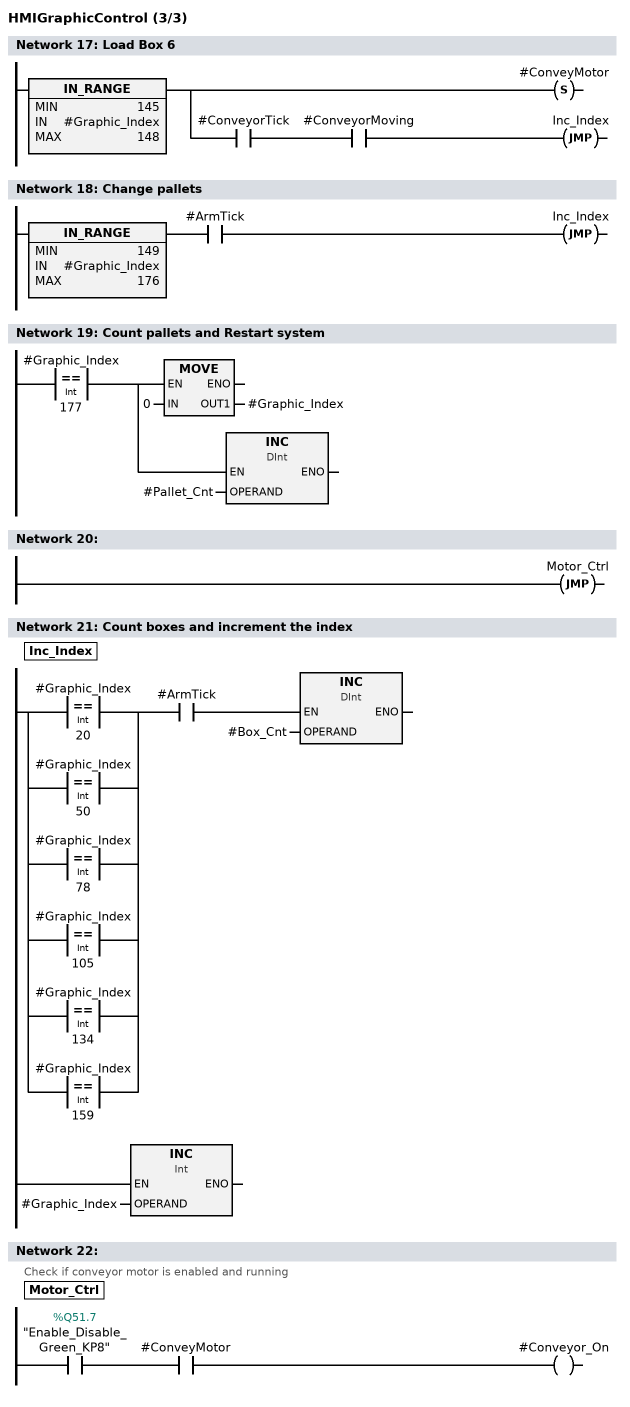
   RUNG wire#powerrail
      { S7_Templates := "SrcType := Int" } InRange(min := 145, in := #Graphic_Index, max := 148)
      wire#w1
      S_Coil( #ConveyMotor )
   END_RUNG
   RUNG wire#w1
      Contact( #ConveyorTick )
      Contact( #ConveyorMoving )
      JumpCoil( Inc_Index )
   END_RUNG
   // the same network as SCL:
   #_w1 := (145 <= #Graphic_Index) AND (#Graphic_Index <= 148);
   IF #_w1 THEN #ConveyMotor := TRUE; END_IF;
   IF #_w1 AND #ConveyorTick AND #ConveyorMoving THEN GOTO Inc_Index; END_IF;
END_REGION

REGION Network 18: Change pallets
   RUNG wire#powerrail
      { S7_Templates := "SrcType := Int" } InRange(min := 149, in := #Graphic_Index, max := 176)
      Contact( #ArmTick )
      JumpCoil( Inc_Index )
   END_RUNG
   // the same network as SCL:
   IF (149 <= #Graphic_Index) AND (#Graphic_Index <= 176) AND #ArmTick THEN GOTO Inc_Index; END_IF;
END_REGION

REGION Network 19: Count pallets and Restart system
   RUNG wire#powerrail
      { S7_Templates := "SrcType := Int" } EQ_Contact(in1 := #Graphic_Index, in2 := 177)
      wire#w1
      Move(in := 0, out1 => #Graphic_Index)
   END_RUNG
   RUNG wire#w1
      { S7_Templates := "DestType := DInt" } Inc( #Pallet_Cnt )
   END_RUNG
   // the same network as SCL:
   #_w1 := #Graphic_Index = 177;
   IF #_w1 THEN
       #Graphic_Index := 0;
       #Pallet_Cnt := #Pallet_Cnt + 1;
   END_IF;
END_REGION

REGION Network 20
   RUNG wire#powerrail
      JumpCoil( Motor_Ctrl )
   END_RUNG
   // the same network as SCL:
   GOTO Motor_Ctrl;
END_REGION

REGION Network 21: Count boxes and increment the index
   Label( Inc_Index )
   RUNG wire#powerrail
      { S7_Templates := "SrcType := Int" } EQ_Contact(in1 := #Graphic_Index, in2 := 20)
      wire#w1
      Contact( #ArmTick )
      { S7_Templates := "DestType := DInt" } Inc( #Box_Cnt )
   END_RUNG
   RUNG wire#powerrail
      { S7_Templates := "SrcType := Int" } EQ_Contact(in1 := #Graphic_Index, in2 := 50)
   END_RUNG wire#w1
   RUNG wire#powerrail
      { S7_Templates := "SrcType := Int" } EQ_Contact(in1 := #Graphic_Index, in2 := 78)
   END_RUNG wire#w1
   RUNG wire#powerrail
      { S7_Templates := "SrcType := Int" } EQ_Contact(in1 := #Graphic_Index, in2 := 105)
   END_RUNG wire#w1
   RUNG wire#powerrail
      { S7_Templates := "SrcType := Int" } EQ_Contact(in1 := #Graphic_Index, in2 := 134)
   END_RUNG wire#w1
   RUNG wire#powerrail
      { S7_Templates := "SrcType := Int" } EQ_Contact(in1 := #Graphic_Index, in2 := 159)
   END_RUNG wire#w1
   RUNG wire#powerrail
      { S7_Templates := "DestType := Int" } Inc( #Graphic_Index )
   END_RUNG
   // the same network as SCL:
   Inc_Index:
   IF ((#Graphic_Index = 20) OR (#Graphic_Index = 50) OR (#Graphic_Index = 78) OR (#Graphic_Index = 105) OR (#Graphic_Index = 134) OR (#Graphic_Index = 159)) AND #ArmTick THEN
       #Box_Cnt := #Box_Cnt + 1;
   END_IF;
   #Graphic_Index := #Graphic_Index + 1;
END_REGION

REGION Network 22
   // Check if conveyor motor is enabled and running
   Label( Motor_Ctrl )
   RUNG wire#powerrail
      Contact( "Enable_Disable_Green_KP8" )
      Contact( #ConveyMotor )
      Coil( #Conveyor_On )
   END_RUNG
   // the same network as SCL:
   Motor_Ctrl:
   #Conveyor_On := "Enable_Disable_Green_KP8" AND #ConveyMotor;
END_REGION
END_FUNCTION_BLOCK

FUNCTION_BLOCK "RPM_to_MPM"   // FB22, LAD
{ S7_Optimized_Access := 'TRUE' }
// stored: AutoNumber false, MemoryReserve 100, SetENOAutomatically false
   VAR_INPUT
      RPM : LReal;
      Diameter : LReal;
   END_VAR
   VAR_OUTPUT
      MRM : Int;   // Input for HMI gauge
   END_VAR
BEGIN

REGION Network 1: Rev Per Minute to Meters Per Minute MRM = (RPM * Diameter) * Pi
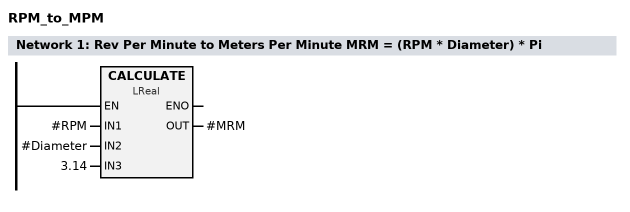
   RUNG wire#powerrail
      { S7_Templates := "SrcType := LReal"; S7_Expression := "(IN2*IN3)*IN1" } Calculate(in1 := #RPM, in2 := #Diameter, in3 := 3.14, out => #MRM)
   END_RUNG
   // the same network as SCL:
   #MRM := (#Diameter*3.14)*#RPM;
END_REGION
END_FUNCTION_BLOCK

FUNCTION_BLOCK "BoilerAlarm"   // FB2, LAD
TITLE = Example of a Typed library block
{ S7_Optimized_Access := 'TRUE' }
// stored: MemoryReserve 100, SetENOAutomatically false
   VAR_INPUT
      "Alarm Bit" : Bool;
   END_VAR
   VAR
      Boiler : Program_Alarm;
   END_VAR
   VAR_TEMP
      "Return" : Int;
      "Current Time" : DTL;
      Boiler_Error : Bool;
      Boiler_Status : Word;
   END_VAR
BEGIN

REGION Network 1
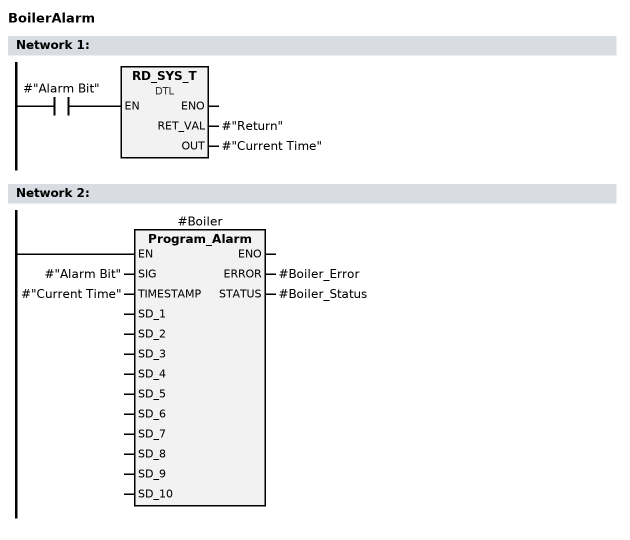
   RUNG wire#powerrail
      Contact( #"Alarm Bit" )
      { S7_Templates := "date_type := DTL" } RD_SYS_T(RET_VAL => #"Return", OUT => #"Current Time")
   END_RUNG
   // the same network as SCL:
   IF #"Alarm Bit" THEN #"Return" := RD_SYS_T(OUT => #"Current Time"); END_IF;
END_REGION

REGION Network 2
   RUNG wire#powerrail
      #Boiler.Program_Alarm(SIG := #"Alarm Bit", TIMESTAMP := #"Current Time", SD_1 :=, SD_2 :=, SD_3 :=, SD_4 :=, SD_5 :=, SD_6 :=, SD_7 :=, SD_8 :=, SD_9 :=, SD_10 :=, Error => #Boiler_Error, Status => #Boiler_Status)
   END_RUNG
   // the same network as SCL:
   #Boiler(SIG := #"Alarm Bit", TIMESTAMP := #"Current Time", Error => #Boiler_Error, Status => #Boiler_Status);   // Program_Alarm
END_REGION
END_FUNCTION_BLOCK

FUNCTION "TimeZone" : Void   // FC4, LAD
{ S7_Optimized_Access := 'TRUE' }
// stored: SetENOAutomatically false
   VAR_IN_OUT
      Zone : "Time Zone";
   END_VAR
   VAR_TEMP
      RealTime : Time;
   END_VAR
   VAR_TEMP   // added for the SCL form of the ladder/FBD networks
      _w1 : Bool;
   END_VAR
BEGIN

REGION Network 1
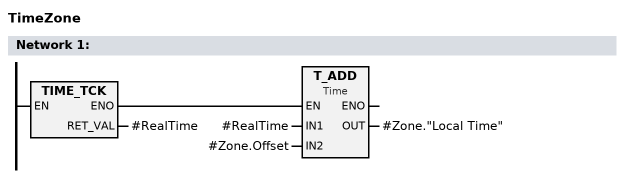
   RUNG wire#powerrail
      TIME_TCK(RET_VAL => #RealTime)
      { S7_Templates := "[date_type := Time, time_type := Time]" } T_ADD(IN1 := #RealTime, IN2 := #Zone.Offset, OUT => #Zone."Local Time")
   END_RUNG
   // the same network as SCL:
   #RealTime := TIME_TCK(ENO => #_w1);
   IF #_w1 THEN T_ADD(IN1 := #RealTime, IN2 := #Zone.Offset, OUT => #Zone."Local Time"); END_IF;
END_REGION
END_FUNCTION

ORGANIZATION_BLOCK "Main_hw"   // OB124, LAD, ProgramCycle
TITLE = "Main Program Sweep (Cycle)"
{ S7_Optimized_Access := 'TRUE' }
// stored: SetENOAutomatically false
   VAR_INPUT
      Initial_Call : Bool;   // Initial call of this OB
      Remanence : Bool;   // =True, if remanent data are available
   END_VAR
   VAR_TEMP   // added for the SCL form of the ladder/FBD networks
      _w1 : Bool;
      _w2 : Bool;
   END_VAR
BEGIN

REGION Network 1: HMI hardware test screen control
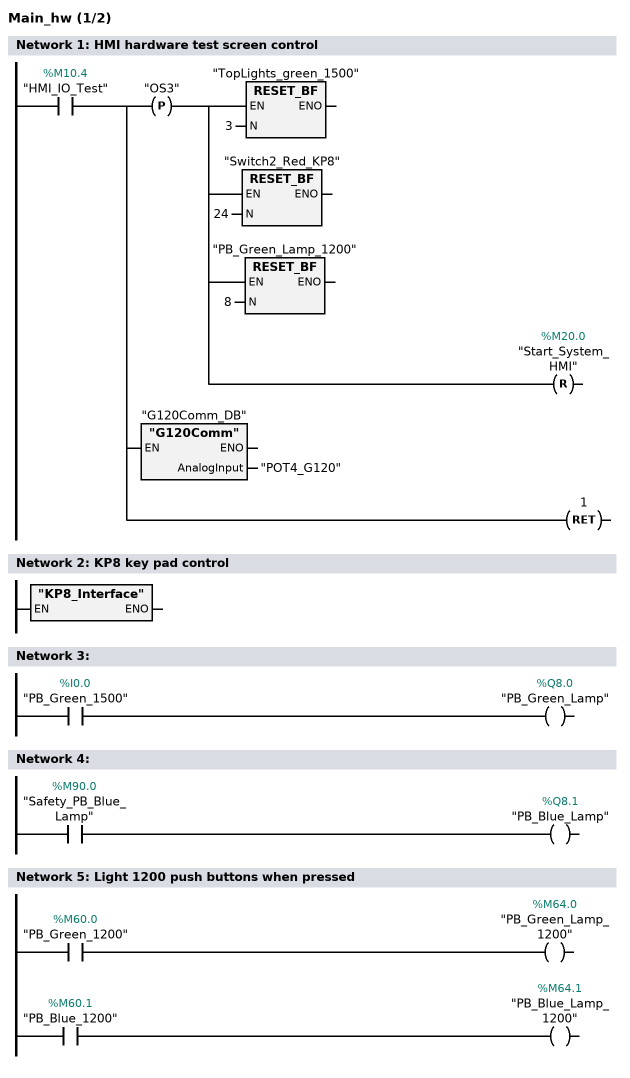
   // no SCL statement known for RBitfield: written as a call
   #_w1 := "HMI_IO_Test" AND NOT "OS3";   // rising edge
   "OS3" := "HMI_IO_Test";
   #_w2 := "HMI_IO_Test";
   IF #_w1 THEN
       RESET_BF(operand := "TopLights_green_1500", n := 3);
       RESET_BF(operand := "Switch2_Red_KP8", n := 24);
       RESET_BF(operand := "PB_Green_Lamp_1200", n := 8);
       "Start_System_HMI" := FALSE;
   END_IF;
   IF #_w2 THEN
       "G120Comm_DB"(AnalogInput => "POT4_G120");   // "G120Comm"
       ENO := 1;
       RETURN;
   END_IF;
END_REGION

REGION Network 2: KP8 key pad control
   RUNG wire#powerrail
      "KP8_Interface"()
   END_RUNG
   // the same network as SCL:
   "KP8_Interface"();
END_REGION

REGION Network 3
   RUNG wire#powerrail
      Contact( "PB_Green_1500" )
      Coil( "PB_Green_Lamp" )
   END_RUNG
   // the same network as SCL:
   "PB_Green_Lamp" := "PB_Green_1500";
END_REGION

REGION Network 4
   RUNG wire#powerrail
      Contact( "Safety_PB_Blue_Lamp" )
      Coil( "PB_Blue_Lamp" )
   END_RUNG
   // the same network as SCL:
   "PB_Blue_Lamp" := "Safety_PB_Blue_Lamp";
END_REGION

REGION Network 5: Light 1200 push buttons when pressed
   RUNG wire#powerrail
      Contact( "PB_Green_1200" )
      Coil( "PB_Green_Lamp_1200" )
   END_RUNG
   RUNG wire#powerrail
      Contact( "PB_Blue_1200" )
      Coil( "PB_Blue_Lamp_1200" )
   END_RUNG
   // the same network as SCL:
   "PB_Green_Lamp_1200" := "PB_Green_1200";
   "PB_Blue_Lamp_1200" := "PB_Blue_1200";
END_REGION

REGION Network 6
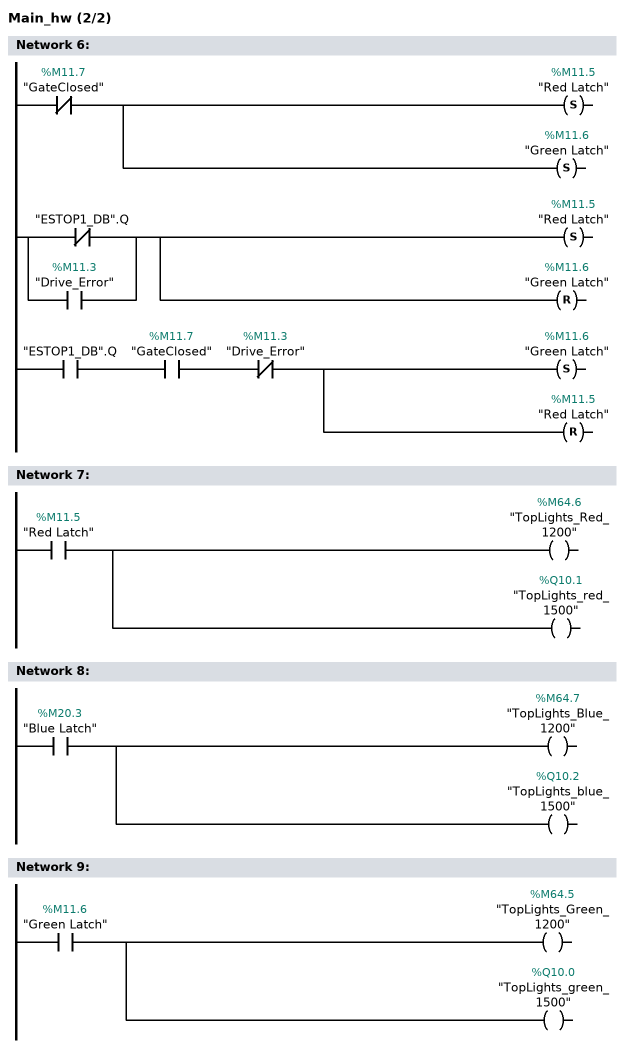
   RUNG wire#powerrail
      I_Contact( "GateClosed" )
      wire#w1
      S_Coil( "Red Latch" )
   END_RUNG
   RUNG wire#w1
      S_Coil( "Green Latch" )
   END_RUNG
   RUNG wire#powerrail
      I_Contact( "ESTOP1_DB".Q )
      wire#w2
      S_Coil( "Red Latch" )
   END_RUNG
   RUNG wire#powerrail
      Contact( "Drive_Error" )
   END_RUNG wire#w2
   RUNG wire#w2
      R_Coil( "Green Latch" )
   END_RUNG
   RUNG wire#powerrail
      Contact( "ESTOP1_DB".Q )
      Contact( "GateClosed" )
      I_Contact( "Drive_Error" )
      wire#w3
      S_Coil( "Green Latch" )
   END_RUNG
   RUNG wire#w3
      R_Coil( "Red Latch" )
   END_RUNG
   // the same network as SCL:
   IF NOT "GateClosed" THEN
       "Red Latch" := TRUE;
       "Green Latch" := TRUE;
   END_IF;
   IF NOT "ESTOP1_DB".Q OR "Drive_Error" THEN
       "Red Latch" := TRUE;
       "Green Latch" := FALSE;
   END_IF;
   IF "ESTOP1_DB".Q AND "GateClosed" AND NOT "Drive_Error" THEN
       "Green Latch" := TRUE;
       "Red Latch" := FALSE;
   END_IF;
END_REGION

REGION Network 7
   RUNG wire#powerrail
      Contact( "Red Latch" )
      wire#w1
      Coil( "TopLights_Red_1200" )
   END_RUNG
   RUNG wire#w1
      Coil( "TopLights_red_1500" )
   END_RUNG
   // the same network as SCL:
   "TopLights_Red_1200" := "Red Latch";
   "TopLights_red_1500" := "Red Latch";
END_REGION

REGION Network 8
   RUNG wire#powerrail
      Contact( "Blue Latch" )
      wire#w1
      Coil( "TopLights_Blue_1200" )
   END_RUNG
   RUNG wire#w1
      Coil( "TopLights_blue_1500" )
   END_RUNG
   // the same network as SCL:
   "TopLights_Blue_1200" := "Blue Latch";
   "TopLights_blue_1500" := "Blue Latch";
END_REGION

REGION Network 9
   RUNG wire#powerrail
      Contact( "Green Latch" )
      wire#w1
      Coil( "TopLights_Green_1200" )
   END_RUNG
   RUNG wire#w1
      Coil( "TopLights_green_1500" )
   END_RUNG
   // the same network as SCL:
   "TopLights_Green_1200" := "Green Latch";
   "TopLights_green_1500" := "Green Latch";
END_REGION
END_ORGANIZATION_BLOCK

FUNCTION_BLOCK "G120Comm"   // FB5, LAD
TITLE = Example of way to read and write the records in the G120
{ S7_Optimized_Access := 'TRUE' }
// stored: MemoryReserve 100, SetENOAutomatically false
   VAR_OUTPUT
      AnalogInput : Real;   // %
   END_VAR
   VAR
      WRREC_Instance { S7_SetPoint := 'True'} : WRREC;
      RDREC_Instance { S7_SetPoint := 'True'} : RDREC;
      WriteRecord : Struct
         Static_1 { S7_SetPoint := 'True'} : "HEADER";
         Static_2 { S7_SetPoint := 'True'} : "PARAMETERADDR";
      END_STRUCT;
      ReadRecord : Struct
         data : Array[0..5] of Byte;
         Value : Real;
      END_STRUCT;
   END_VAR
   // WriteRecord.Static_1.REQ_REF := 1;
   // WriteRecord.Static_1.REQ_ID := 1;
   // WriteRecord.Static_1.AXIS := 1;
   // WriteRecord.Static_1.NO_PARAM := 1;
   // WriteRecord.Static_2.ATTRIBUTE := 16;
   // WriteRecord.Static_2.NO_ELEM := 1;
   // WriteRecord.Static_2.PARA_NO := 755;
   // WriteRecord.Static_2.SUBINDEX := 0;
BEGIN
END_FUNCTION_BLOCK

FUNCTION "KP8_Interface" : Void   // FC3, LAD
TITLE = Control Lights on the KP8
{ S7_Optimized_Access := 'TRUE' }
// stored: SetENOAutomatically false
   VAR_TEMP
      RetVal : Int;
      Color : Int;
      ColorStop : Int;
      ColorRun : Int;
   END_VAR
   VAR CONSTANT
      Addr : Int := 50;   // Starting Q address of the KP8
      Off : Int;   // Color
      Red : Int := 1;   // Color
      Yellow : Int := 2;   // Color
      Green : Int := 3;   // Color
      Blue : Int := 4;   // Color
      White : Int := 5;   // Color
      Switch2 : Int := 0;
      JogFwd : Int := 1;
      Stop : Int := 2;
      Reset : Int := 3;
      Switch1 : Int := 4;
      JogRev : Int := 5;
      Run : Int := 6;
      Enable : Int := 7;
   END_VAR
   VAR_TEMP   // added for the SCL form of the ladder/FBD networks
      _w1 : Bool;
      _w2 : Bool;
   END_VAR
BEGIN

REGION Network 1
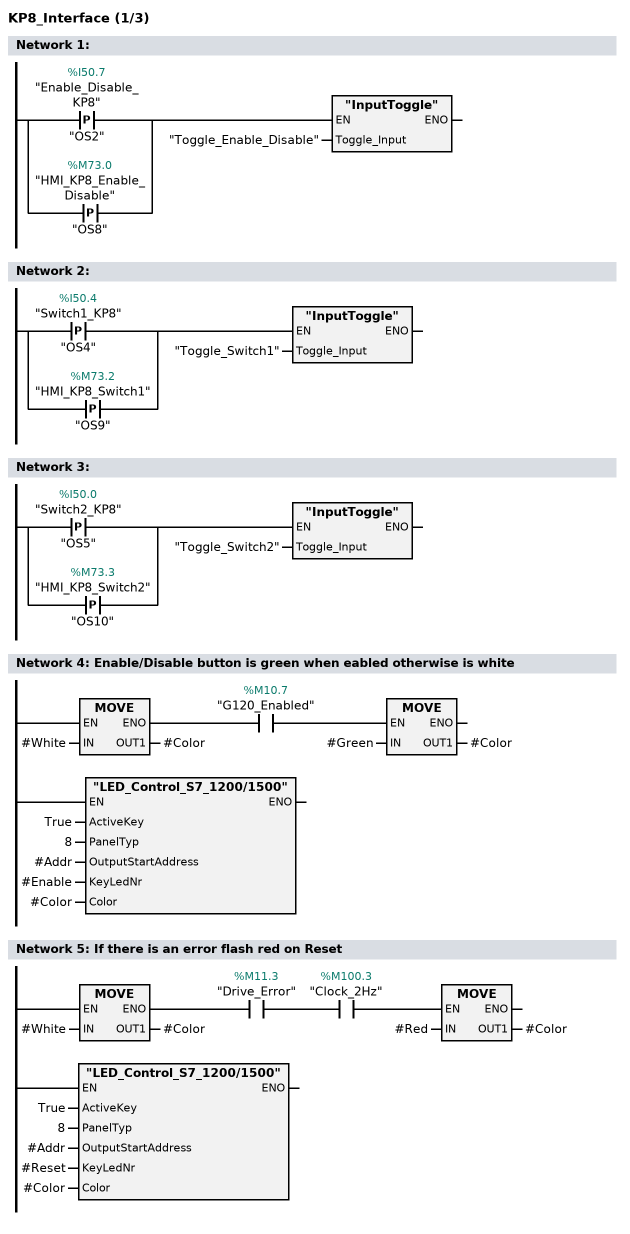
   RUNG wire#powerrail
      P_Contact(operand := "Enable_Disable_KP8", bit := "OS2")
      wire#w1
      "InputToggle"(Toggle_Input := "Toggle_Enable_Disable")
   END_RUNG
   RUNG wire#powerrail
      P_Contact(operand := "HMI_KP8_Enable_Disable", bit := "OS8")
   END_RUNG wire#w1
   // the same network as SCL:
   #_w1 := "Enable_Disable_KP8" AND NOT "OS2";   // rising edge of "Enable_Disable_KP8"
   "OS2" := "Enable_Disable_KP8";
   #_w2 := "HMI_KP8_Enable_Disable" AND NOT "OS8";   // rising edge of "HMI_KP8_Enable_Disable"
   "OS8" := "HMI_KP8_Enable_Disable";
   IF #_w1 OR #_w2 THEN "InputToggle"(Toggle_Input := "Toggle_Enable_Disable"); END_IF;
END_REGION

REGION Network 2
   RUNG wire#powerrail
      P_Contact(operand := "Switch1_KP8", bit := "OS4")
      wire#w1
      "InputToggle"(Toggle_Input := "Toggle_Switch1")
   END_RUNG
   RUNG wire#powerrail
      P_Contact(operand := "HMI_KP8_Switch1", bit := "OS9")
   END_RUNG wire#w1
   // the same network as SCL:
   #_w1 := "Switch1_KP8" AND NOT "OS4";   // rising edge of "Switch1_KP8"
   "OS4" := "Switch1_KP8";
   #_w2 := "HMI_KP8_Switch1" AND NOT "OS9";   // rising edge of "HMI_KP8_Switch1"
   "OS9" := "HMI_KP8_Switch1";
   IF #_w1 OR #_w2 THEN "InputToggle"(Toggle_Input := "Toggle_Switch1"); END_IF;
END_REGION

REGION Network 3
   RUNG wire#powerrail
      P_Contact(operand := "Switch2_KP8", bit := "OS5")
      wire#w1
      "InputToggle"(Toggle_Input := "Toggle_Switch2")
   END_RUNG
   RUNG wire#powerrail
      P_Contact(operand := "HMI_KP8_Switch2", bit := "OS10")
   END_RUNG wire#w1
   // the same network as SCL:
   #_w1 := "Switch2_KP8" AND NOT "OS5";   // rising edge of "Switch2_KP8"
   "OS5" := "Switch2_KP8";
   #_w2 := "HMI_KP8_Switch2" AND NOT "OS10";   // rising edge of "HMI_KP8_Switch2"
   "OS10" := "HMI_KP8_Switch2";
   IF #_w1 OR #_w2 THEN "InputToggle"(Toggle_Input := "Toggle_Switch2"); END_IF;
END_REGION

REGION Network 4: Enable/Disable button is green when eabled otherwise is white
   RUNG wire#powerrail
      Move(in := #White, out1 => #Color)
      Contact( "G120_Enabled" )
      Move(in := #Green, out1 => #Color)
   END_RUNG
   RUNG wire#powerrail
      "LED_Control_S7_1200/1500"(ActiveKey := True, PanelTyp := 8, OutputStartAddress := #Addr, KeyLedNr := #Enable, Color := #Color)
   END_RUNG
   // the same network as SCL:
   #Color := #White;
   IF "G120_Enabled" THEN #Color := #Green; END_IF;
   "LED_Control_S7_1200/1500"(ActiveKey := True,
                           PanelTyp := 8,
                           OutputStartAddress := #Addr,
                           KeyLedNr := #Enable,
                           Color := #Color);
END_REGION

REGION Network 5: If there is an error flash red on Reset
   RUNG wire#powerrail
      Move(in := #White, out1 => #Color)
      Contact( "Drive_Error" )
      Contact( "Clock_2Hz" )
      Move(in := #Red, out1 => #Color)
   END_RUNG
   RUNG wire#powerrail
      "LED_Control_S7_1200/1500"(ActiveKey := True, PanelTyp := 8, OutputStartAddress := #Addr, KeyLedNr := #Reset, Color := #Color)
   END_RUNG
   // the same network as SCL:
   #Color := #White;
   IF "Drive_Error" AND "Clock_2Hz" THEN #Color := #Red; END_IF;
   "LED_Control_S7_1200/1500"(ActiveKey := True,
                           PanelTyp := 8,
                           OutputStartAddress := #Addr,
                           KeyLedNr := #Reset,
                           Color := #Color);
END_REGION

REGION Network 6: Run and Stop
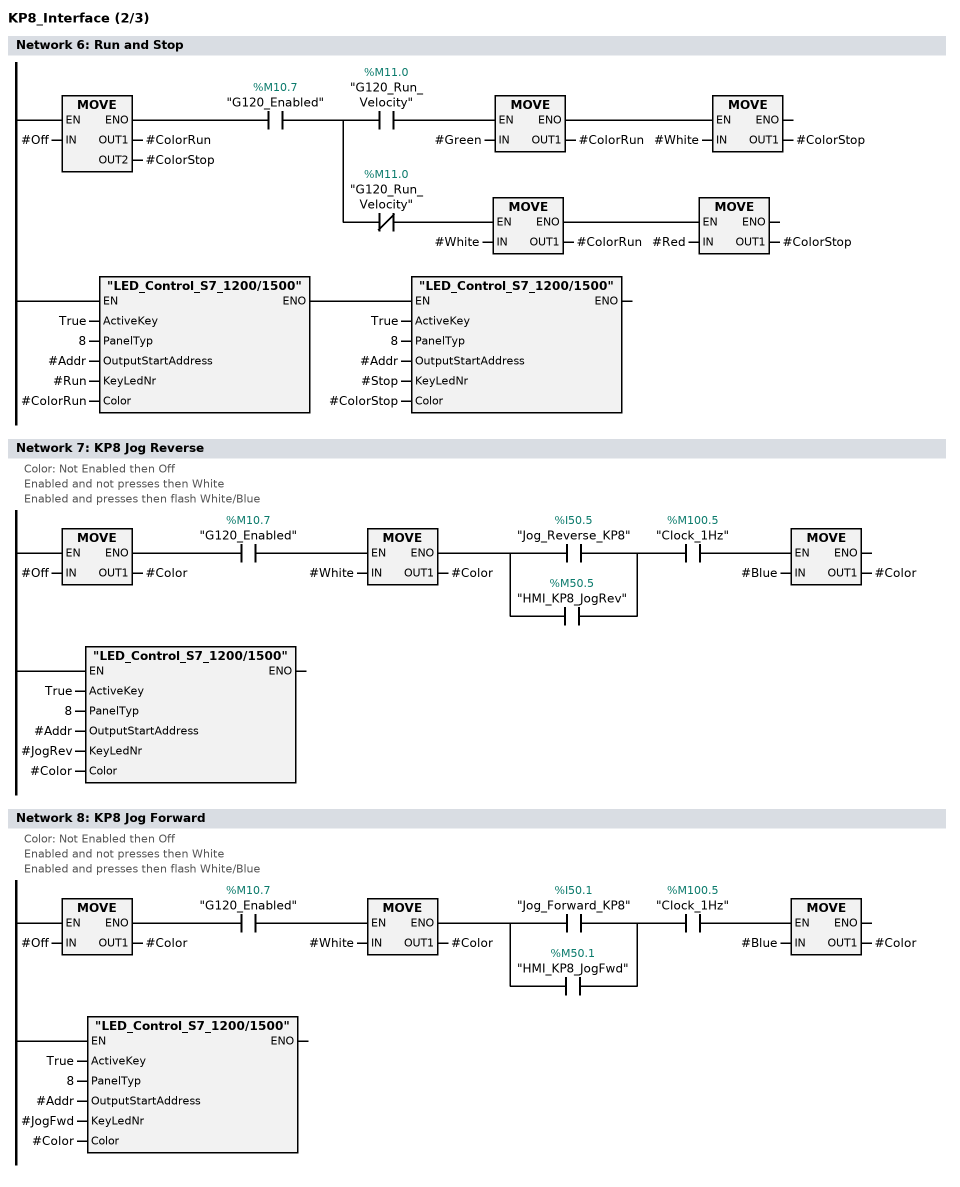
   RUNG wire#powerrail
      Move(in := #Off, out1 => #ColorRun, out2 => #ColorStop)
      Contact( "G120_Enabled" )
      wire#w1
      Contact( "G120_Run_Velocity" )
      Move(in := #Green, out1 => #ColorRun)
      Move(in := #White, out1 => #ColorStop)
   END_RUNG
   RUNG wire#w1
      I_Contact( "G120_Run_Velocity" )
      Move(in := #White, out1 => #ColorRun)
      Move(in := #Red, out1 => #ColorStop)
   END_RUNG
   RUNG wire#powerrail
      "LED_Control_S7_1200/1500"(ActiveKey := True, PanelTyp := 8, OutputStartAddress := #Addr, KeyLedNr := #Run, Color := #ColorRun)
      "LED_Control_S7_1200/1500"(ActiveKey := True, PanelTyp := 8, OutputStartAddress := #Addr, KeyLedNr := #Stop, Color := #ColorStop)
   END_RUNG
   // the same network as SCL:
   #ColorRun := #Off;
   #ColorStop := #Off;
   IF "G120_Enabled" AND "G120_Run_Velocity" THEN
       #ColorRun := #Green;
       #ColorStop := #White;
   END_IF;
   IF "G120_Enabled" AND NOT "G120_Run_Velocity" THEN
       #ColorRun := #White;
       #ColorStop := #Red;
   END_IF;
   "LED_Control_S7_1200/1500"(ActiveKey := True,
                           PanelTyp := 8,
                           OutputStartAddress := #Addr,
                           KeyLedNr := #Run,
                           Color := #ColorRun,
                           ENO => #_w1);
   IF #_w1 THEN
       "LED_Control_S7_1200/1500"(ActiveKey := True,
                               PanelTyp := 8,
                               OutputStartAddress := #Addr,
                               KeyLedNr := #Stop,
                               Color := #ColorStop);
   END_IF;
END_REGION

REGION Network 7: KP8 Jog Reverse
   // Color: Not Enabled then Off
   //             Enabled and not presses then White
   //             Enabled and presses then flash White/Blue
   RUNG wire#powerrail
      Move(in := #Off, out1 => #Color)
      Contact( "G120_Enabled" )
      Move(in := #White, out1 => #Color)
      wire#w1
      Contact( "Jog_Reverse_KP8" )
      wire#w2
      Contact( "Clock_1Hz" )
      Move(in := #Blue, out1 => #Color)
   END_RUNG
   RUNG wire#w1
      Contact( "HMI_KP8_JogRev" )
   END_RUNG wire#w2
   RUNG wire#powerrail
      "LED_Control_S7_1200/1500"(ActiveKey := True, PanelTyp := 8, OutputStartAddress := #Addr, KeyLedNr := #JogRev, Color := #Color)
   END_RUNG
   // the same network as SCL:
   #Color := #Off;
   IF "G120_Enabled" THEN #Color := #White; END_IF;
   IF "G120_Enabled" AND ("Jog_Reverse_KP8" OR "HMI_KP8_JogRev") AND "Clock_1Hz" THEN
       #Color := #Blue;
   END_IF;
   "LED_Control_S7_1200/1500"(ActiveKey := True,
                           PanelTyp := 8,
                           OutputStartAddress := #Addr,
                           KeyLedNr := #JogRev,
                           Color := #Color);
END_REGION

REGION Network 8: KP8 Jog Forward
   // Color: Not Enabled then Off
   //             Enabled and not presses then White
   //             Enabled and presses then flash White/Blue
   RUNG wire#powerrail
      Move(in := #Off, out1 => #Color)
      Contact( "G120_Enabled" )
      Move(in := #White, out1 => #Color)
      wire#w1
      Contact( "Jog_Forward_KP8" )
      wire#w2
      Contact( "Clock_1Hz" )
      Move(in := #Blue, out1 => #Color)
   END_RUNG
   RUNG wire#w1
      Contact( "HMI_KP8_JogFwd" )
   END_RUNG wire#w2
   RUNG wire#powerrail
      "LED_Control_S7_1200/1500"(ActiveKey := True, PanelTyp := 8, OutputStartAddress := #Addr, KeyLedNr := #JogFwd, Color := #Color)
   END_RUNG
   // the same network as SCL:
   #Color := #Off;
   IF "G120_Enabled" THEN #Color := #White; END_IF;
   IF "G120_Enabled" AND ("Jog_Forward_KP8" OR "HMI_KP8_JogFwd") AND "Clock_1Hz" THEN
       #Color := #Blue;
   END_IF;
   "LED_Control_S7_1200/1500"(ActiveKey := True,
                           PanelTyp := 8,
                           OutputStartAddress := #Addr,
                           KeyLedNr := #JogFwd,
                           Color := #Color);
END_REGION

REGION Network 9: KP8 Switch 1
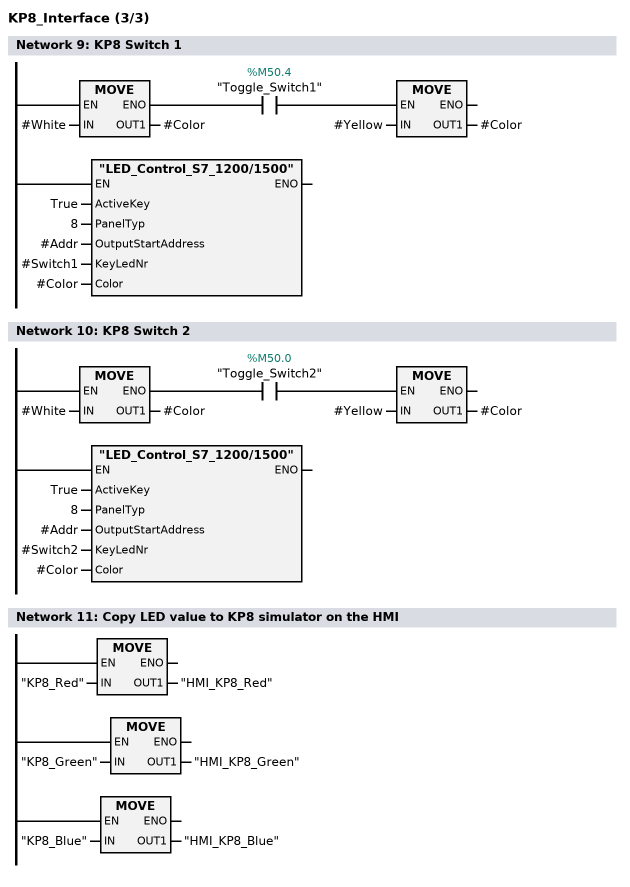
   RUNG wire#powerrail
      Move(in := #White, out1 => #Color)
      Contact( "Toggle_Switch1" )
      Move(in := #Yellow, out1 => #Color)
   END_RUNG
   RUNG wire#powerrail
      "LED_Control_S7_1200/1500"(ActiveKey := True, PanelTyp := 8, OutputStartAddress := #Addr, KeyLedNr := #Switch1, Color := #Color)
   END_RUNG
   // the same network as SCL:
   #Color := #White;
   IF "Toggle_Switch1" THEN #Color := #Yellow; END_IF;
   "LED_Control_S7_1200/1500"(ActiveKey := True,
                           PanelTyp := 8,
                           OutputStartAddress := #Addr,
                           KeyLedNr := #Switch1,
                           Color := #Color);
END_REGION

REGION Network 10: KP8 Switch 2
   RUNG wire#powerrail
      Move(in := #White, out1 => #Color)
      Contact( "Toggle_Switch2" )
      Move(in := #Yellow, out1 => #Color)
   END_RUNG
   RUNG wire#powerrail
      "LED_Control_S7_1200/1500"(ActiveKey := True, PanelTyp := 8, OutputStartAddress := #Addr, KeyLedNr := #Switch2, Color := #Color)
   END_RUNG
   // the same network as SCL:
   #Color := #White;
   IF "Toggle_Switch2" THEN #Color := #Yellow; END_IF;
   "LED_Control_S7_1200/1500"(ActiveKey := True,
                           PanelTyp := 8,
                           OutputStartAddress := #Addr,
                           KeyLedNr := #Switch2,
                           Color := #Color);
END_REGION

REGION Network 11: Copy LED value to KP8 simulator on the HMI
   RUNG wire#powerrail
      Move(in := "KP8_Red", out1 => "HMI_KP8_Red")
   END_RUNG
   RUNG wire#powerrail
      Move(in := "KP8_Green", out1 => "HMI_KP8_Green")
   END_RUNG
   RUNG wire#powerrail
      Move(in := "KP8_Blue", out1 => "HMI_KP8_Blue")
   END_RUNG
   // the same network as SCL:
   "HMI_KP8_Red" := "KP8_Red";
   "HMI_KP8_Green" := "KP8_Green";
   "HMI_KP8_Blue" := "KP8_Blue";
END_REGION
END_FUNCTION

FUNCTION "InputToggle" : Void   // FC2, LAD
{ S7_Optimized_Access := 'TRUE' }
// stored: SetENOAutomatically false
   VAR_IN_OUT
      Toggle_Input : Bool;
   END_VAR
BEGIN

REGION Network 1
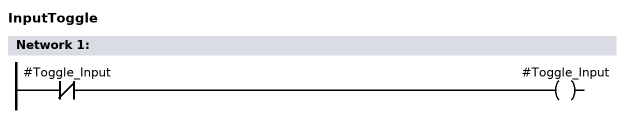
   RUNG wire#powerrail
      I_Contact( #Toggle_Input )
      Coil( #Toggle_Input )
   END_RUNG
   // the same network as SCL:
   #Toggle_Input := NOT #Toggle_Input;
END_REGION
END_FUNCTION

ORGANIZATION_BLOCK "TestCallEnv"   // OB10000, FBD, ProgramCycle
TITLE = "Main Program Sweep (Cycle)"
{ S7_Optimized_Access := 'TRUE' }
// #@AutoGenerated
// stored: SetENOAutomatically false
   VAR_INPUT
      Initial_Call : Bool;   // Initial call of this OB
      Remanence : Bool;   // =True, if remanent data are available
   END_VAR
BEGIN

REGION Network 1: : Call LPythagorean - AppTest LPythagoreanTestCase
   // #@AutoGenerated
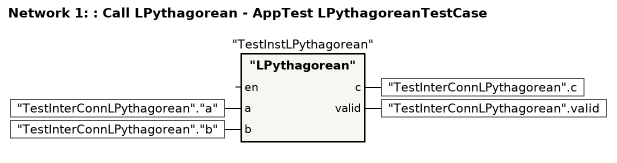
   "TestInstLPythagorean"("a" := "TestInterConnLPythagorean"."a",   // "LPythagorean"
                          "b" := "TestInterConnLPythagorean"."b",
                          c => "TestInterConnLPythagorean".c,
                          valid => "TestInterConnLPythagorean".valid);
END_REGION
END_ORGANIZATION_BLOCK

FUNCTION_BLOCK "LPythagorean"
{ S7_Optimized_Access := 'TRUE' }
VERSION : 0.1
   VAR_INPUT 
      a : Real;
      b : Real;
   END_VAR

   VAR_OUTPUT 
      c : Real;
      valid : Bool;
   END_VAR


BEGIN
	IF #a >= 0 AND #b >= 0 THEN
	    #c := SQRT(#a * #a + #b * #b);  // Calculate the hypotenuse
	    #valid := TRUE;
	ELSE
	    #c := -1;  // Invalid input, set c to -1
	    #valid := FALSE;
	END_IF;
	
END_FUNCTION_BLOCK

FUNCTION_BLOCK "Main_Safety_RTG1"   // FB, F_LAD
{ S7_Optimized_Access := 'TRUE' }
// stored: AutoNumber false
BEGIN

REGION Network 1
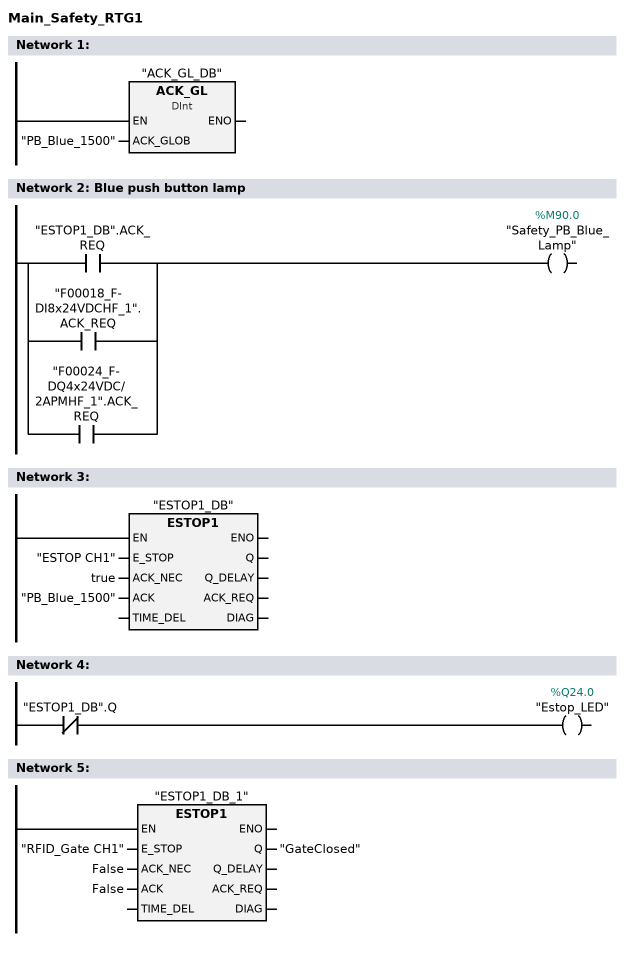
   RUNG wire#powerrail
      { S7_Templates := "codedbool_type := DInt" } "ACK_GL_DB".ACK_GL(ACK_GLOB := "PB_Blue_1500")
   END_RUNG
   // the same network as SCL:
   "ACK_GL_DB"(ACK_GLOB := "PB_Blue_1500");   // ACK_GL
END_REGION

REGION Network 2: Blue push button lamp
   RUNG wire#powerrail
      Contact( "ESTOP1_DB".ACK_REQ )
      wire#w1
      Coil( "Safety_PB_Blue_Lamp" )
   END_RUNG
   RUNG wire#powerrail
      Contact( "F00018_F-DI8x24VDCHF_1".ACK_REQ )
   END_RUNG wire#w1
   RUNG wire#powerrail
      Contact( "F00024_F-DQ4x24VDC/2APMHF_1".ACK_REQ )
   END_RUNG wire#w1
   // the same network as SCL:
   "Safety_PB_Blue_Lamp" := "ESTOP1_DB".ACK_REQ OR "F00018_F-DI8x24VDCHF_1".ACK_REQ OR "F00024_F-DQ4x24VDC/2APMHF_1".ACK_REQ;
END_REGION

REGION Network 3
   RUNG wire#powerrail
      "ESTOP1_DB".ESTOP1(E_STOP := "ESTOP CH1", ACK_NEC := true, ACK := "PB_Blue_1500", TIME_DEL :=, Q =>, Q_DELAY =>, ACK_REQ =>, DIAG =>)
   END_RUNG
   // the same network as SCL:
   "ESTOP1_DB"(E_STOP := "ESTOP CH1", ACK_NEC := true, ACK := "PB_Blue_1500");   // ESTOP1
END_REGION

REGION Network 4
   RUNG wire#powerrail
      I_Contact( "ESTOP1_DB".Q )
      Coil( "Estop_LED" )
   END_RUNG
   // the same network as SCL:
   "Estop_LED" := NOT "ESTOP1_DB".Q;
END_REGION

REGION Network 5
   RUNG wire#powerrail
      "ESTOP1_DB_1".ESTOP1(E_STOP := "RFID_Gate CH1", ACK_NEC := False, ACK := False, TIME_DEL :=, Q => "GateClosed", Q_DELAY =>, ACK_REQ =>, DIAG =>)
   END_RUNG
   // the same network as SCL:
   "ESTOP1_DB_1"(E_STOP := "RFID_Gate CH1", ACK_NEC := False, ACK := False, Q => "GateClosed");   // ESTOP1
END_REGION
END_FUNCTION_BLOCK

FUNCTION_BLOCK "StartStop"
{ S7_Optimized_Access := 'TRUE' }
VERSION : 0.1
   VAR_INPUT 
      start : Bool;
   END_VAR

   VAR_OUTPUT 
      status : Bool;
   END_VAR


BEGIN
	IF #start THEN
	    #status := True;
	ELSE
	    #status := False;
	END_IF;
	
END_FUNCTION_BLOCK

DATA_BLOCK "Boiler_1"   // DB11
// stored: InstanceOfName BoilerAlarm, InstanceOfType FB
"BoilerAlarm"
BEGIN
END_DATA_BLOCK

DATA_BLOCK "Boiler_2"   // DB12
// stored: InstanceOfName BoilerAlarm, InstanceOfType FB
"BoilerAlarm"
BEGIN
END_DATA_BLOCK

DATA_BLOCK "LPythagorean_DB"   // DB3
// stored: InstanceOfName LPythagorean, InstanceOfType FB
"LPythagorean"
BEGIN
END_DATA_BLOCK

DATA_BLOCK "Main_Safety_RTG1_DB"   // DB18, F_DB
// stored: AutoNumber false, InstanceOfName Main_Safety_RTG1, InstanceOfType FB
"Main_Safety_RTG1"
BEGIN
END_DATA_BLOCK

DATA_BLOCK "StartStop_DB"   // DB4
// stored: InstanceOfName StartStop, InstanceOfType FB
"StartStop"
BEGIN
END_DATA_BLOCK

DATA_BLOCK "ARM_RPM_to_MPM_DB"   // DB23
// stored: AutoNumber false, InstanceOfName RPM_to_MPM, InstanceOfType FB
"RPM_to_MPM"
BEGIN
END_DATA_BLOCK

DATA_BLOCK "Conveyor_RPM_to_MPM_DB"   // DB22
// stored: AutoNumber false, InstanceOfName RPM_to_MPM, InstanceOfType FB
"RPM_to_MPM"
BEGIN
END_DATA_BLOCK

DATA_BLOCK "HMIGraphicControl_DB"   // DB21
// stored: AutoNumber false, InstanceOfName HMIGraphicControl, InstanceOfType FB
"HMIGraphicControl"
BEGIN
END_DATA_BLOCK

DATA_BLOCK "TestInstLPythagorean"   // DB10002
// #@AutoGenerated
// stored: InstanceOfName LPythagorean, InstanceOfType FB
"LPythagorean"
BEGIN
END_DATA_BLOCK

DATA_BLOCK "1200Comm_DB"   // DB2
// stored: InstanceOfName 1200Comm, InstanceOfType FB
"1200Comm"
BEGIN
END_DATA_BLOCK

DATA_BLOCK "G120Comm_DB"   // DB17
// stored: InstanceOfName G120Comm, InstanceOfType FB
"G120Comm"
BEGIN
END_DATA_BLOCK

DATA_BLOCK "SpeedAxis_1"   // DB3, Motion_DB
// stored: InstanceOfName TO_SpeedAxis, OfSystemLibElement TO_SpeedAxis, OfSystemLibVersion 8.0
TO_SpeedAxis   // technology object, version 8.0
   // // inherited from TO_Axis
   // // inherited from TO_Object
   // VAR
   //    Velocity { ExternalWritable := 'False'} : LReal;
   //    Acceleration { ExternalWritable := 'False'} : LReal;
   //    ActualSpeed { ExternalWritable := 'False'} : LReal;
   //    VelocitySetpoint { ExternalWritable := 'False'} : LReal;
   //    Actor { S7_SetPoint := 'True'} : TO_Struct_Actor;
   //    TorqueLimiting { S7_SetPoint := 'True'} : TO_Struct_TorqueLimiting;
   //    LoadGear { S7_SetPoint := 'True'} : TO_Struct_LoadGear;
   //    DynamicLimits { S7_SetPoint := 'True'} : TO_Struct_DynamicLimits;
   //    DynamicDefaults { S7_SetPoint := 'True'} : TO_Struct_DynamicDefaults;
   //    Override { S7_SetPoint := 'True'} : TO_Struct_Override;
   //    Units { ExternalWritable := 'False'; S7_SetPoint := 'True'} : TO_Struct_Units;
   //    StatusDrive { ExternalWritable := 'False'; S7_SetPoint := 'True'} : TO_Struct_StatusDrive;
   //    StatusTorqueData { ExternalWritable := 'False'; S7_SetPoint := 'True'} : TO_Struct_StatusTorqueData;
   //    StatusMotionIn { ExternalWritable := 'False'; S7_SetPoint := 'True'} : TO_Struct_StatusMotionIn;
   //    StatusInterpreterMotion { ExternalWritable := 'False'; S7_SetPoint := 'True'} : TO_Struct_StatusInterpreterMotion;
   //    StatusWord { ExternalWritable := 'False'} : DWord;
   //    StatusWord2 { ExternalWritable := 'False'} : DWord;
   //    ErrorWord { ExternalWritable := 'False'} : DWord;
   //    ErrorDetail { ExternalWritable := 'False'; S7_SetPoint := 'True'} : TO_Struct_ErrorDetail;
   //    WarningWord { ExternalWritable := 'False'} : DWord;
   //    ControlPanel { S7_SetPoint := 'True'} : TO_Struct_ControlPanel;
   //    InternalToTrace { S7_SetPoint := 'True'} : Array[1..4] of TO_Struct_Internal;
   //    VirtualAxis { ExternalWritable := 'False'; S7_SetPoint := 'True'} : TO_Struct_VirtualAxis;
   //    Simulation { S7_SetPoint := 'True'} : TO_Struct_AxisSimulation;
   // END_VAR
BEGIN
   Actor.Interface.AddressIn.RID := 16#2080708;
   Actor.Interface.AddressOut.RID := 16#2080709;
   Actor.DriveParameter.ReferenceSpeed := 1500.0;
   Actor.DriveParameter.MaxSpeed := 1500.0;
   DynamicLimits.MaxVelocity := 1500.0;
   DynamicLimits.MaxAcceleration := 500.0;
   DynamicLimits.MaxDeceleration := 500.0;
   DynamicLimits.MaxJerk := 10000.0;
   DynamicDefaults.Acceleration := 200.0;
   DynamicDefaults.Deceleration := 200.0;
   DynamicDefaults.Jerk := 4000.0;
   DynamicDefaults.EmergencyDeceleration := 500.0;
   VirtualAxis.Mode := 1;
   VirtualAxis.Mode := 1;
   _Actor.Interface.Telegram := 1;
END_DATA_BLOCK
